KUKA KRL program: MyProgram_067().src

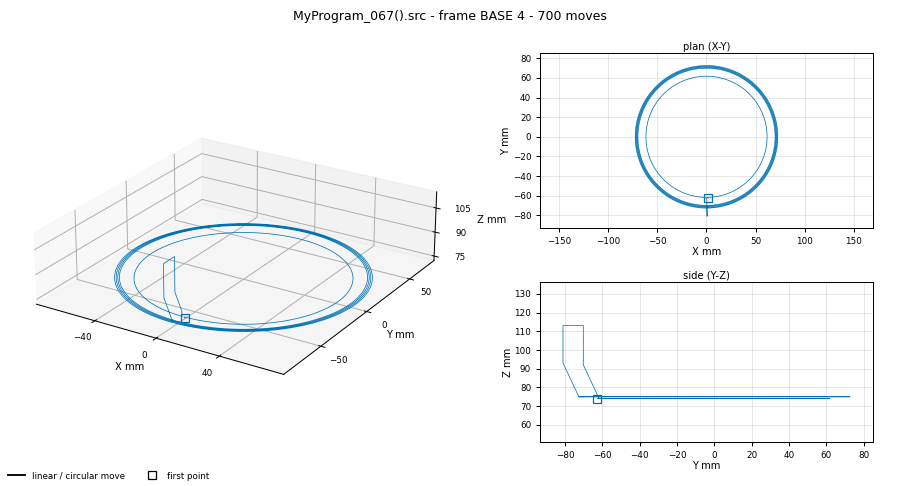
[picture p0: tool path of MyProgram_067().src in frame BASE 4, 700 of 700 moves have a stored position in this frame; points joined in program order, loops and branches not executed]
&ACCESS RVP
&REL 1
&PARAM TEMPLATE = C:\KRC\Roboter\Template\vorgabe
&PARAM EDITMASK = *
DEF MyProgram_067()
; ---- Setting reference (Base) ----
$BASE = BASE_DATA[4]

; --------------------------
; ---- Setting tool (TCP) ----
$TOOL = TOOL_DATA[3]
; --------------------------

$VEL.CP = VEL_APROX_PRINT
Startdeposition()
$VEL.CP = VEL_PRINT
LIN {X 1.6603,Y -62.6279,Z 74,A -94.6717,B 24.8978,C -2.3339,E1 25.0027,E2 178.7795} C_DIS
LIN {X 1.6603,Y -62.6279,Z 74,A -94.6717,B 24.8978,C -2.3339,E1 25.0027,E2 178.7795} C_DIS
Enddeposition()
LIN {X 0.3854,Y -61.7225,Z 74,A -95.5899,B 24.8959,C -2.3553,E1 25.0003,E2 179.6469} C_DIS
Startdeposition()
$VEL.CP = VEL_PRINT
LIN {X 2.2389,Y -61.6864,Z 74,A -92.854,B 24.8939,C -2.3781,E1 25.0081,E2 176.8573} C_DIS
LIN {X 5.2551,Y -61.5029,Z 74,A -90.0412,B 24.8937,C -2.3796,E1 25.0159,E2 174.0424} C_DIS
LIN {X 8.2959,Y -61.1671,Z 74,A -87.2156,B 24.8937,C -2.381,E1 25.0237,E2 171.2156} C_DIS
LIN {X 11.2776,Y -60.6881,Z 74,A -84.42,B 24.8934,C -2.383,E1 25.0314,E2 168.4183} C_DIS
LIN {X 14.2593,Y -60.0576,Z 74,A -81.5934,B 24.8932,C -2.3855,E1 25.0391,E2 165.5894} C_DIS
LIN {X 17.1475,Y -59.2974,Z 74,A -78.8211,B 24.8929,C -2.3885,E1 25.0466,E2 162.8146} C_DIS
LIN {X 20.0481,Y -58.3806,Z 74,A -76.0037,B 24.8927,C -2.3917,E1 25.0541,E2 159.9949} C_DIS
LIN {X 22.9015,Y -57.3215,Z 74,A -73.1974,B 24.8923,C -2.3951,E1 25.0614,E2 157.1866} C_DIS
LIN {X 25.6576,Y -56.1417,Z 74,A -70.4181,B 24.892,C -2.3992,E1 25.0685,E2 154.4046} C_DIS
LIN {X 28.3851,Y -54.8133,Z 74,A -67.6066,B 24.8916,C -2.4037,E1 25.0755,E2 151.5901} C_DIS
LIN {X 31.0814,Y -53.3309,Z 74,A -64.7699,B 24.8912,C -2.4082,E1 25.0824,E2 148.751} C_DIS
LIN {X 33.6554,Y -51.7451,Z 74,A -61.9856,B 24.8907,C -2.413,E1 25.089,E2 145.9645} C_DIS
LIN {X 35.9087,Y -50.2063,Z 74,A -59.347,B 24.89,C -2.4206,E1 25.0951,E2 143.3169} C_DIS
LIN {X 37.9795,Y -48.66,Z 74,A -57.0724,B 24.8899,C -2.4227,E1 25.1001,E2 141.0458} C_DIS
LIN {X 40.2995,Y -46.7566,Z 74,A -54.2947,B 24.8893,C -2.4286,E1 25.106,E2 138.2646} C_DIS
LIN {X 42.5511,Y -44.7173,Z 74,A -51.4857,B 24.8887,C -2.4349,E1 25.1118,E2 135.4522} C_DIS
LIN {X 44.6978,Y -42.5717,Z 74,A -48.6871,B 24.8881,C -2.4413,E1 25.1172,E2 132.6505} C_DIS
LIN {X 46.7261,Y -40.3349,Z 74,A -45.9001,B 24.8875,C -2.448,E1 25.1224,E2 129.8602} C_DIS
LIN {X 48.6424,Y -38.0018,Z 74,A -43.1096,B 24.8869,C -2.455,E1 25.1273,E2 127.0662} C_DIS
LIN {X 50.471,Y -35.5376,Z 74,A -40.2933,B 24.8862,C -2.4619,E1 25.1319,E2 124.2472} C_DIS
LIN {X 52.1299,Y -33.0559,Z 74,A -37.5283,B 24.8855,C -2.4694,E1 25.1361,E2 121.4782} C_DIS
LIN {X 53.7046,Y -30.4313,Z 74,A -34.7004,B 24.8848,C -2.4772,E1 25.1401,E2 118.6466} C_DIS
LIN {X 55.1351,Y -27.7556,Z 74,A -31.916,B 24.8841,C -2.4846,E1 25.1437,E2 115.8594} C_DIS
LIN {X 56.4098,Y -25.0629,Z 74,A -29.1531,B 24.8834,C -2.4927,E1 25.1469,E2 113.0922} C_DIS
LIN {X 57.5735,Y -22.2598,Z 74,A -26.3562,B 24.8826,C -2.5007,E1 25.1498,E2 110.2918} C_DIS
LIN {X 58.5947,Y -19.4131,Z 74,A -23.5811,B 24.8819,C -2.5085,E1 25.1523,E2 107.514} C_DIS
LIN {X 59.4511,Y -16.6049,Z 74,A -20.9319,B 24.8813,C -2.5151,E1 25.1544,E2 104.8645} C_DIS
LIN {X 60.0566,Y -14.2635,Z 74,A -18.6458,B 24.8805,C -2.5231,E1 25.1559,E2 102.5726} C_DIS
LIN {X 60.6831,Y -11.3049,Z 74,A -15.8403,B 24.8797,C -2.5319,E1 25.1574,E2 99.7627} C_DIS
LIN {X 61.1664,Y -8.3014,Z 74,A -13.0483,B 24.8789,C -2.54,E1 25.1586,E2 96.9679} C_DIS
LIN {X 61.4957,Y -5.3376,Z 74,A -10.2981,B 24.8781,C -2.5483,E1 25.1593,E2 94.2143} C_DIS
LIN {X 61.6847,Y -2.2864,Z 74,A -7.4845,B 24.8773,C -2.5567,E1 25.1597,E2 91.3975} C_DIS
LIN {X 61.7226,Y 0.753,Z 74,A -4.6831,B 24.8765,C -2.5652,E1 25.1597,E2 88.5929} C_DIS
LIN {X 61.613,Y 3.7495,Z 74,A -1.9141,B 24.8757,C -2.5736,E1 25.1594,E2 85.8205} C_DIS
LIN {X 61.3515,Y 6.7991,Z 74,A 0.9072,B 24.8748,C -2.582,E1 25.1586,E2 82.9961} C_DIS
LIN {X 60.9452,Y 9.7941,Z 74,A 3.6994,B 24.874,C -2.5903,E1 25.1574,E2 80.2006} C_DIS
LIN {X 60.3961,Y 12.7486,Z 74,A 6.4727,B 24.8732,C -2.5985,E1 25.1559,E2 77.4242} C_DIS
LIN {X 59.69,Y 15.7273,Z 74,A 9.2777,B 24.8725,C -2.6061,E1 25.154,E2 74.6173} C_DIS
LIN {X 58.8596,Y 18.5946,Z 74,A 12.0434,B 24.8717,C -2.6142,E1 25.1518,E2 71.8482} C_DIS
LIN {X 57.8593,Y 21.507,Z 74,A 14.8896,B 24.8709,C -2.6222,E1 25.1491,E2 68.9991} C_DIS
LIN {X 56.7304,Y 24.3291,Z 74,A 17.68,B 24.8702,C -2.6295,E1 25.1461,E2 66.2068} C_DIS
LIN {X 55.4727,Y 27.0745,Z 74,A 20.4596,B 24.8695,C -2.6366,E1 25.1428,E2 63.4253} C_DIS
LIN {X 54.1001,Y 29.7219,Z 74,A 23.2284,B 24.8687,C -2.6441,E1 25.1391,E2 60.6533} C_DIS
LIN {X 52.5629,Y 32.3632,Z 74,A 26.0462,B 24.868,C -2.6511,E1 25.1351,E2 57.8335} C_DIS
LIN {X 50.9005,Y 34.9197,Z 74,A 28.8466,B 24.8674,C -2.6574,E1 25.1307,E2 55.032} C_DIS
LIN {X 49.1544,Y 37.3371,Z 74,A 31.6173,B 24.8667,C -2.6642,E1 25.1261,E2 52.2586} C_DIS
LIN {X 47.2479,Y 39.7224,Z 74,A 34.4307,B 24.8661,C -2.6703,E1 25.1211,E2 49.4438} C_DIS
LIN {X 45.245,Y 41.9895,Z 74,A 37.2149,B 24.8655,C -2.6759,E1 25.1159,E2 46.6586} C_DIS
LIN {X 43.1689,Y 44.1207,Z 74,A 39.9738,B 24.865,C -2.6816,E1 25.1105,E2 43.8978} C_DIS
LIN {X 40.866,Y 46.2623,Z 74,A 42.8566,B 24.8645,C -2.6865,E1 25.1045,E2 41.0151} C_DIS
LIN {X 38.5801,Y 48.1852,Z 74,A 45.6354,B 24.8639,C -2.6918,E1 25.0985,E2 38.2344} C_DIS
LIN {X 36.1981,Y 49.9991,Z 74,A 48.4152,B 24.8634,C -2.6966,E1 25.0923,E2 35.4531} C_DIS
LIN {X 33.6858,Y 51.7251,Z 74,A 51.2263,B 24.863,C -2.7006,E1 25.0857,E2 32.6418} C_DIS
LIN {X 31.0844,Y 53.3292,Z 74,A 54.0465,B 24.8626,C -2.7044,E1 25.079,E2 29.8214} C_DIS
LIN {X 28.4548,Y 54.7773,Z 74,A 56.8332,B 24.8623,C -2.7081,E1 25.0721,E2 27.034} C_DIS
LIN {X 25.7053,Y 56.1203,Z 74,A 59.6662,B 24.862,C -2.7112,E1 25.065,E2 24.2008} C_DIS
LIN {X 22.9276,Y 57.3111,Z 74,A 62.4652,B 24.8617,C -2.714,E1 25.0577,E2 21.4018} C_DIS
LIN {X 20.125,Y 58.3541,Z 74,A 65.2331,B 24.8614,C -2.7162,E1 25.0505,E2 18.6341} C_DIS
LIN {X 17.2286,Y 59.2739,Z 74,A 68.0604,B 24.8612,C -2.7184,E1 25.0429,E2 15.8067} C_DIS
LIN {X 14.2598,Y 60.0575,Z 74,A 70.8892,B 24.8611,C -2.7196,E1 25.0353,E2 12.9792} C_DIS
LIN {X 11.3005,Y 60.684,Z 74,A 73.7045,B 24.861,C -2.721,E1 25.0275,E2 10.1642} C_DIS
LIN {X 8.3143,Y 61.1646,Z 74,A 76.5104,B 24.8609,C -2.7217,E1 25.0198,E2 7.3591} C_DIS
LIN {X 5.3318,Y 61.4963,Z 74,A 79.2951,B 24.8609,C -2.722,E1 25.0121,E2 4.5754} C_DIS
LIN {X 2.2751,Y 61.6852,Z 74,A 82.1298,B 24.8609,C -2.7217,E1 25.0042,E2 1.7423} C_DIS
LIN {X -0.7492,Y 61.7226,Z 74,A 84.9385,B 24.8609,C -2.7212,E1 24.9963,E2 -1.0651} C_DIS
LIN {X -3.7534,Y 61.6128,Z 74,A 87.7403,B 24.861,C -2.7205,E1 24.9885,E2 -3.8658} C_DIS
LIN {X -6.8036,Y 61.3511,Z 74,A 90.5853,B 24.8611,C -2.7191,E1 24.9806,E2 -6.7091} C_DIS
LIN {X -9.7997,Y 60.9443,Z 74,A 93.3961,B 24.8613,C -2.7173,E1 24.9729,E2 -9.5181} C_DIS
LIN {X -12.7347,Y 60.399,Z 74,A 96.1815,B 24.8615,C -2.7154,E1 24.9652,E2 -12.3021} C_DIS
LIN {X -15.7307,Y 59.6891,Z 74,A 99.0339,B 24.8618,C -2.7126,E1 24.9575,E2 -15.1517} C_DIS
LIN {X -18.6193,Y 58.8519,Z 74,A 101.8354,B 24.8621,C -2.7097,E1 24.95,E2 -17.9511} C_DIS
LIN {X -21.5107,Y 57.8579,Z 74,A 104.6799,B 24.8625,C -2.7063,E1 24.9426,E2 -20.7932} C_DIS
LIN {X -24.3152,Y 56.7364,Z 74,A 107.495,B 24.8628,C -2.7026,E1 24.9353,E2 -23.6059} C_DIS
LIN {X -27.0608,Y 55.4793,Z 74,A 110.298,B 24.8633,C -2.6983,E1 24.9282,E2 -26.4059} C_DIS
LIN {X -29.7396,Y 54.0905,Z 74,A 113.118,B 24.8637,C -2.6941,E1 24.9213,E2 -29.2236} C_DIS
LIN {X -32.3962,Y 52.5425,Z 74,A 115.9816,B 24.8642,C -2.6891,E1 24.9144,E2 -32.0842} C_DIS
LIN {X -34.9253,Y 50.8966,Z 74,A 118.787,B 24.8647,C -2.6839,E1 24.9079,E2 -34.8863} C_DIS
LIN {X -37.3715,Y 49.1285,Z 74,A 121.6084,B 24.8653,C -2.6785,E1 24.9016,E2 -37.705} C_DIS
LIN {X -39.7131,Y 47.2556,Z 74,A 124.4197,B 24.8658,C -2.6731,E1 24.8956,E2 -40.514} C_DIS
LIN {X -42.02,Y 45.2168,Z 74,A 127.2728,B 24.8665,C -2.6665,E1 24.8897,E2 -43.3628} C_DIS
LIN {X -44.1641,Y 43.125,Z 74,A 130.0821,B 24.8671,C -2.6605,E1 24.8841,E2 -46.1696} C_DIS
LIN {X -46.2286,Y 40.9042,Z 74,A 132.9067,B 24.8678,C -2.6537,E1 24.8788,E2 -48.9906} C_DIS
LIN {X -48.1786,Y 38.5882,Z 74,A 135.7462,B 24.8684,C -2.6471,E1 24.8738,E2 -51.8273} C_DIS
LIN {X -50.0053,Y 36.1897,Z 74,A 138.5606,B 24.8691,C -2.6399,E1 24.8691,E2 -54.6383} C_DIS
LIN {X -51.7358,Y 33.6696,Z 74,A 141.4276,B 24.8699,C -2.6327,E1 24.8647,E2 -57.5024} C_DIS
LIN {X -53.3279,Y 31.0865,Z 74,A 144.2266,B 24.8707,C -2.6245,E1 24.8607,E2 -60.2961} C_DIS
LIN {X -54.7373,Y 28.5307,Z 74,A 146.9486,B 24.8714,C -2.6169,E1 24.8571,E2 -63.0145} C_DIS
LIN {X -56.0379,Y 25.8822,Z 74,A 149.7819,B 24.872,C -2.6106,E1 24.8537,E2 -65.8481} C_DIS
LIN {X -57.3141,Y 22.9202,Z 74,A 152.7404,B 24.873,C -2.601,E1 24.8505,E2 -68.8} C_DIS
LIN {X -58.3546,Y 20.1234,Z 74,A 155.5303,B 24.8738,C -2.593,E1 24.8479,E2 -71.5865} C_DIS
LIN {X -59.2693,Y 17.2441,Z 74,A 158.3637,B 24.8746,C -2.5849,E1 24.8456,E2 -74.4169} C_DIS
LIN {X -60.0108,Y 14.4512,Z 74,A 161.1191,B 24.8752,C -2.5779,E1 24.8437,E2 -77.1716} C_DIS
LIN {X -60.6856,Y 11.2914,Z 74,A 164.0763,B 24.8762,C -2.5677,E1 24.8421,E2 -80.122} C_DIS
LIN {X -61.1659,Y 8.3053,Z 74,A 166.9043,B 24.877,C -2.5592,E1 24.841,E2 -82.9465} C_DIS
LIN {X -61.4958,Y 5.3368,Z 74,A 169.6974,B 24.8779,C -2.5508,E1 24.8402,E2 -85.7364} C_DIS
LIN {X -61.6838,Y 2.3093,Z 74,A 172.5358,B 24.8787,C -2.5423,E1 24.8398,E2 -88.5716} C_DIS
LIN {X -61.7234,Y -0.6427,Z 74,A 174.9824,B 24.88,C -2.5283,E1 24.8398,E2 -90.9993} C_DIS
LIN {X -61.6544,Y -2.9918,Z 74,A 177.5004,B 24.88,C -2.5276,E1 24.8401,E2 -93.5309} C_DIS
LIN {X -61.4303,Y -6.0469,Z 74,A -179.6505,B 24.8809,C -2.5188,E1 24.8408,E2 -96.376} C_DIS
LIN {X -61.0638,Y -9.0239,Z 74,A -176.8408,B 24.8817,C -2.5106,E1 24.8418,E2 -99.183} C_DIS
LIN {X -60.5483,Y -12.0051,Z 74,A -174.0035,B 24.8824,C -2.5026,E1 24.8433,E2 -102.0179} C_DIS
LIN {X -59.8873,Y -14.9575,Z 74,A -171.1785,B 24.8832,C -2.4944,E1 24.8451,E2 -104.8399} C_DIS
LIN {X -59.0657,Y -17.9298,Z 74,A -168.3034,B 24.884,C -2.4861,E1 24.8473,E2 -107.7118} C_DIS
LIN {X -58.1191,Y -20.7947,Z 74,A -165.4927,B 24.8847,C -2.4781,E1 24.8499,E2 -110.5194} C_DIS
LIN {X -57.0415,Y -23.59,Z 74,A -162.6844,B 24.8854,C -2.4707,E1 24.8528,E2 -113.3257} C_DIS
LIN {X -55.8177,Y -26.3552,Z 74,A -159.8503,B 24.8861,C -2.4634,E1 24.8561,E2 -116.1578} C_DIS
LIN {X -54.4463,Y -29.0833,Z 74,A -157.0013,B 24.8868,C -2.456,E1 24.8597,E2 -119.0044} C_DIS
LIN {X -52.9641,Y -31.702,Z 74,A -154.1929,B 24.8874,C -2.449,E1 24.8637,E2 -121.8106} C_DIS
LIN {X -51.3391,Y -34.2714,Z 74,A -151.3597,B 24.8881,C -2.4421,E1 24.868,E2 -124.6415} C_DIS
LIN {X -49.6548,Y -36.6683,Z 74,A -148.7218,B 24.8888,C -2.4339,E1 24.8723,E2 -127.2727} C_DIS
LIN {X -47.9584,Y -38.8599,Z 74,A -146.0482,B 24.8892,C -2.4299,E1 24.8769,E2 -129.9492} C_DIS
LIN {X -45.9944,Y -41.1657,Z 74,A -143.4282,B 24.8901,C -2.4198,E1 24.8817,E2 -132.5572} C_DIS
LIN {X -44.1975,Y -43.0907,Z 74,A -140.7574,B 24.8901,C -2.419,E1 24.8869,E2 -135.2376} C_DIS
LIN {X -42.0309,Y -45.2066,Z 74,A -137.9338,B 24.8907,C -2.4136,E1 24.8926,E2 -138.06} C_DIS
LIN {X -39.7422,Y -47.2314,Z 74,A -135.0869,B 24.8911,C -2.4084,E1 24.8986,E2 -140.9056} C_DIS
LIN {X -37.3852,Y -49.118,Z 74,A -132.2786,B 24.8916,C -2.4036,E1 24.9048,E2 -143.7127} C_DIS
LIN {X -34.9404,Y -50.8862,Z 74,A -129.4612,B 24.892,C -2.3994,E1 24.9112,E2 -146.5297} C_DIS
LIN {X -32.3849,Y -52.5496,Z 74,A -126.6115,B 24.8923,C -2.3955,E1 24.9179,E2 -149.3793} C_DIS
LIN {X -29.7939,Y -54.0606,Z 74,A -123.8249,B 24.8927,C -2.3918,E1 24.9247,E2 -152.1652} C_DIS
LIN {X -27.1134,Y -55.4534,Z 74,A -121.0032,B 24.8929,C -2.3887,E1 24.9317,E2 -154.9871} C_DIS
LIN {X -24.3297,Y -56.7301,Z 74,A -118.1616,B 24.8932,C -2.3856,E1 24.939,E2 -157.8282} C_DIS
LIN {X -21.5259,Y -57.8521,Z 74,A -115.3559,B 24.8934,C -2.3831,E1 24.9463,E2 -160.6338} C_DIS
LIN {X -18.6841,Y -58.8313,Z 74,A -112.5554,B 24.8936,C -2.3811,E1 24.9537,E2 -163.4348} C_DIS
LIN {X -15.7315,Y -59.6889,Z 74,A -109.7003,B 24.8938,C -2.3794,E1 24.9614,E2 -166.2902} C_DIS
LIN {X -12.8257,Y -60.3798,Z 74,A -106.9156,B 24.8938,C -2.3783,E1 24.969,E2 -169.076} C_DIS
LIN {X -9.8156,Y -60.9417,Z 74,A -104.0755,B 24.8939,C -2.3774,E1 24.9768,E2 -171.9166} C_DIS
LIN {X -6.804,Y -61.3511,Z 74,A -101.2661,B 24.894,C -2.3767,E1 24.9846,E2 -174.7263} C_DIS
LIN {X -3.8288,Y -61.6081,Z 74,A -98.4765,B 24.894,C -2.3771,E1 24.9924,E2 -177.518} C_DIS
LIN {X -0.7696,Y -61.7223,Z 74,A -95.6423,B 24.894,C -2.3773,E1 25.0003,E2 -180.3531} C_DIS
LIN {X -0.7696,Y -61.7223,Z 74,A -95.6423,B 24.894,C -2.3773,E1 25.0003,E2 -180.3531} C_DIS
Enddeposition()
LIN {X 0.385,Y -63.8356,Z 78.5315,A -95.5798,B 24.8963,C -2.351,E1 25.0003,E2 -180.3531} C_DIS
LIN {X 0.384,Y -70.1749,Z 92.1262,A -95.5544,B 24.8972,C -2.3403,E1 25.0003,E2 -180.3531} C_DIS
LIN {X 0.384,Y -70.1749,Z 113.1262,A -95.9113,B 24.8836,C -2.4906,E1 25.0003,E2 -180.3531} C_DIS
LIN {X 0.598,Y -81.0561,Z 113.1262,A -94.7572,B 24.8982,C -2.3288,E1 25.0024,E2 -181.1228} C_DIS
LIN {X 0.598,Y -81.0561,Z 93.1262,A -94.4172,B 24.9104,C -2.1856,E1 25.0024,E2 -181.1228} C_DIS
LIN {X 0.5139,Y -74.7174,Z 79.5315,A -94.4404,B 24.9096,C -2.1954,E1 25.0024,E2 -181.1228} C_DIS
LIN {X 0.4859,Y -72.6045,Z 75,A -94.4497,B 24.9093,C -2.1993,E1 25.0024,E2 -181.1228} C_DIS
Startdeposition()
$VEL.CP = VEL_PRINT
LIN {X -2.6725,Y -72.56,Z 75,A -97.8407,B 24.9112,C -2.1754,E1 24.9928,E2 -177.6748} C_DIS
LIN {X -5.5896,Y -72.3926,Z 75,A -100.1329,B 24.9112,C -2.1757,E1 24.9864,E2 -175.3826} C_DIS
LIN {X -8.6409,Y -72.0921,Z 75,A -102.5384,B 24.9112,C -2.1764,E1 24.9797,E2 -172.9772} C_DIS
LIN {X -11.5346,Y -71.6872,Z 75,A -104.9376,B 24.9113,C -2.1745,E1 24.9731,E2 -170.5715} C_DIS
LIN {X -14.1654,Y -71.214,Z 75,A -107.0488,B 24.9113,C -2.1753,E1 24.9673,E2 -168.4598} C_DIS
LIN {X -16.7769,Y -70.6444,Z 75,A -109.1605,B 24.9112,C -2.1762,E1 24.9616,E2 -166.3476} C_DIS
LIN {X -19.3658,Y -69.979,Z 75,A -111.2729,B 24.9111,C -2.1774,E1 24.9559,E2 -164.2349} C_DIS
LIN {X -21.9284,Y -69.2188,Z 75,A -113.3855,B 24.911,C -2.1788,E1 24.9502,E2 -162.122} C_DIS
LIN {X -24.4613,Y -68.3648,Z 75,A -115.4988,B 24.9108,C -2.1805,E1 24.9447,E2 -160.0085} C_DIS
LIN {X -26.961,Y -67.4181,Z 75,A -117.6126,B 24.9107,C -2.1824,E1 24.9392,E2 -157.8946} C_DIS
LIN {X -29.4242,Y -66.38,Z 75,A -119.5937,B 24.9102,C -2.1877,E1 24.9341,E2 -155.9216} C_DIS
LIN {X -31.8476,Y -65.252,Z 75,A -121.8419,B 24.9103,C -2.1868,E1 24.9284,E2 -153.6654} C_DIS
LIN {X -34.4465,Y -63.9169,Z 75,A -124.0765,B 24.9099,C -2.1915,E1 24.9229,E2 -151.4358} C_DIS
LIN {X -37.1143,Y -62.4056,Z 75,A -126.3435,B 24.9093,C -2.1985,E1 24.9175,E2 -149.1788} C_DIS
LIN {X -39.0552,Y -61.2097,Z 75,A -128.3088,B 24.9094,C -2.1972,E1 24.9128,E2 -147.2042} C_DIS
LIN {X -41.2817,Y -59.7307,Z 75,A -130.4258,B 24.9092,C -2.2004,E1 24.9079,E2 -145.0877} C_DIS
LIN {X -43.4522,Y -58.1708,Z 75,A -132.5433,B 24.9089,C -2.2038,E1 24.9031,E2 -142.9708} C_DIS
LIN {X -45.8694,Y -56.2844,Z 75,A -134.8122,B 24.9082,C -2.2117,E1 24.8982,E2 -140.7123} C_DIS
LIN {X -47.91,Y -54.5579,Z 75,A -136.9308,B 24.9079,C -2.2155,E1 24.8937,E2 -138.5945} C_DIS
LIN {X -49.8857,Y -52.7575,Z 75,A -139.0494,B 24.9076,C -2.2194,E1 24.8893,E2 -136.4767} C_DIS
LIN {X -51.7937,Y -50.8856,Z 75,A -141.1686,B 24.9073,C -2.2236,E1 24.8852,E2 -134.3584} C_DIS
LIN {X -53.6316,Y -48.9447,Z 75,A -143.4337,B 24.9072,C -2.2245,E1 24.8808,E2 -132.0856} C_DIS
LIN {X -55.5582,Y -46.7481,Z 75,A -145.818,B 24.9069,C -2.2279,E1 24.8765,E2 -129.6985} C_DIS
LIN {X -57.3931,Y -44.4743,Z 75,A -148.0842,B 24.9064,C -2.2342,E1 24.8726,E2 -127.4368} C_DIS
LIN {X -59.2196,Y -42.0116,Z 75,A -150.5022,B 24.9059,C -2.2401,E1 24.8686,E2 -125.0212} C_DIS
LIN {X -60.8628,Y -39.5956,Z 75,A -152.9141,B 24.9056,C -2.2435,E1 24.8649,E2 -122.6053} C_DIS
LIN {X -62.4056,Y -37.1143,Z 75,A -155.1552,B 24.9049,C -2.251,E1 24.8616,E2 -120.3705} C_DIS
LIN {X -63.9169,Y -34.4465,Z 75,A -157.5744,B 24.9044,C -2.2574,E1 24.8583,E2 -117.954} C_DIS
LIN {X -65.252,Y -31.8476,Z 75,A -159.9875,B 24.9041,C -2.2613,E1 24.8553,E2 -115.5371} C_DIS
LIN {X -66.38,Y -29.4242,Z 75,A -161.9261,B 24.9032,C -2.271,E1 24.8531,E2 -113.6111} C_DIS
LIN {X -67.4181,Y -26.961,Z 75,A -164.2138,B 24.9031,C -2.273,E1 24.8507,E2 -111.3155} C_DIS
LIN {X -68.4472,Y -24.2265,Z 75,A -166.4758,B 24.9024,C -2.2807,E1 24.8485,E2 -109.059} C_DIS
LIN {X -69.409,Y -21.3151,Z 75,A -168.7509,B 24.9015,C -2.2911,E1 24.8466,E2 -106.7957} C_DIS
LIN {X -70.1465,Y -18.7459,Z 75,A -171.0203,B 24.9013,C -2.2938,E1 24.8449,E2 -104.5197} C_DIS
LIN {X -70.8449,Y -15.9088,Z 75,A -173.435,B 24.9009,C -2.2984,E1 24.8433,E2 -102.1017} C_DIS
LIN {X -71.4266,Y -13.0454,Z 75,A -175.6787,B 24.9002,C -2.3069,E1 24.8421,E2 -99.8649} C_DIS
LIN {X -71.9136,Y -10.0182,Z 75,A -178.1001,B 24.8995,C -2.3143,E1 24.8411,E2 -97.447} C_DIS
LIN {X -72.2596,Y -7.1169,Z 75,A 179.4846,B 24.8991,C -2.3191,E1 24.8404,E2 -95.0286} C_DIS
LIN {X -72.4726,Y -4.4524,Z 75,A 177.4944,B 24.8983,C -2.3283,E1 24.84,E2 -93.0486} C_DIS
LIN {X -72.5873,Y -1.7819,Z 75,A 175.2122,B 24.898,C -2.3312,E1 24.8398,E2 -90.7594} C_DIS
LIN {X -72.5873,Y 1.7819,Z 75,A 172.4034,B 24.8972,C -2.3402,E1 24.8398,E2 -87.9551} C_DIS
LIN {X -72.4726,Y 4.4524,Z 75,A 170.4127,B 24.8964,C -2.3495,E1 24.8402,E2 -85.9747} C_DIS
LIN {X -72.2596,Y 7.1169,Z 75,A 168.1543,B 24.8961,C -2.3529,E1 24.8407,E2 -83.7109} C_DIS
LIN {X -71.9136,Y 10.0182,Z 75,A 165.9103,B 24.8954,C -2.3616,E1 24.8415,E2 -81.4742} C_DIS
LIN {X -71.4266,Y 13.0454,Z 75,A 163.6341,B 24.8944,C -2.3724,E1 24.8426,E2 -79.2103} C_DIS
LIN {X -70.898,Y 15.6656,Z 75,A 161.5098,B 24.8938,C -2.3787,E1 24.8438,E2 -77.0886} C_DIS
LIN {X -70.3937,Y 17.7964,Z 75,A 159.5628,B 24.8938,C -2.3792,E1 24.8451,E2 -75.1315} C_DIS
LIN {X -69.5535,Y 20.8387,Z 75,A 157.2614,B 24.8927,C -2.3911,E1 24.8469,E2 -72.8452} C_DIS
LIN {X -68.83,Y 23.1158,Z 75,A 155.2541,B 24.8924,C -2.3942,E1 24.8486,E2 -70.8338} C_DIS
LIN {X -67.832,Y 25.8989,Z 75,A 152.8679,B 24.8919,C -2.4002,E1 24.8509,E2 -68.4482} C_DIS
LIN {X -66.7361,Y 28.6074,Z 75,A 150.4533,B 24.8915,C -2.4046,E1 24.8535,E2 -66.031} C_DIS
LIN {X -65.5301,Y 31.2688,Z 75,A 148.2102,B 24.8907,C -2.4129,E1 24.8561,E2 -63.7953} C_DIS
LIN {X -64.1516,Y 34.0075,Z 75,A 145.9355,B 24.8898,C -2.4231,E1 24.859,E2 -61.5329} C_DIS
LIN {X -62.8564,Y 36.3457,Z 75,A 143.8125,B 24.8893,C -2.4289,E1 24.8619,E2 -59.4125} C_DIS
LIN {X -61.476,Y 38.6347,Z 75,A 141.7013,B 24.8887,C -2.4347,E1 24.865,E2 -57.3044} C_DIS
LIN {X -60.2328,Y 40.5456,Z 75,A 139.7188,B 24.8887,C -2.4356,E1 24.8681,E2 -55.314} C_DIS
LIN {X -58.4673,Y 43.0524,Z 75,A 137.4451,B 24.8878,C -2.4454,E1 24.8717,E2 -53.0527} C_DIS
LIN {X -56.843,Y 45.1753,Z 75,A 135.3232,B 24.8873,C -2.4506,E1 24.8754,E2 -50.9332} C_DIS
LIN {X -55.3968,Y 46.9375,Z 75,A 133.3533,B 24.8873,C -2.4513,E1 24.8789,E2 -48.9559} C_DIS
LIN {X -53.3657,Y 49.2345,Z 75,A 131.0807,B 24.8864,C -2.4607,E1 24.8831,E2 -46.6956} C_DIS
LIN {X -51.5174,Y 51.1654,Z 75,A 128.8185,B 24.8862,C -2.4623,E1 24.8875,E2 -44.4274} C_DIS
LIN {X -49.4179,Y 53.1974,Z 75,A 126.537,B 24.8857,C -2.4682,E1 24.8921,E2 -42.1506} C_DIS
LIN {X -47.4264,Y 54.9803,Z 75,A 124.331,B 24.8854,C -2.4707,E1 24.8968,E2 -39.9418} C_DIS
LIN {X -45.3705,Y 56.6887,Z 75,A 122.2974,B 24.8848,C -2.477,E1 24.9012,E2 -37.9155} C_DIS
LIN {X -43.2532,Y 58.3203,Z 75,A 120.0445,B 24.8848,C -2.478,E1 24.9062,E2 -35.657} C_DIS
LIN {X -41.0773,Y 59.8728,Z 75,A 117.9258,B 24.8844,C -2.4819,E1 24.911,E2 -33.5405} C_DIS
LIN {X -38.8457,Y 61.3441,Z 75,A 115.8074,B 24.884,C -2.4857,E1 24.916,E2 -31.4242} C_DIS
LIN {X -36.5615,Y 62.7324,Z 75,A 113.6896,B 24.8837,C -2.4893,E1 24.9211,E2 -29.3085} C_DIS
LIN {X -34.0075,Y 64.1516,Z 75,A 111.453,B 24.8832,C -2.4948,E1 24.9266,E2 -27.0787} C_DIS
LIN {X -31.2688,Y 65.5301,Z 75,A 109.1851,B 24.8825,C -2.5022,E1 24.9322,E2 -24.8225} C_DIS
LIN {X -28.8356,Y 66.6367,Z 75,A 107.0687,B 24.8822,C -2.5051,E1 24.9376,E2 -22.7079} C_DIS
LIN {X -26.3633,Y 67.6528,Z 75,A 104.9559,B 24.8819,C -2.5079,E1 24.9431,E2 -20.5971} C_DIS
LIN {X -24.2265,Y 68.4472,Z 75,A 102.9886,B 24.8821,C -2.5061,E1 24.9483,E2 -18.6217} C_DIS
LIN {X -21.3151,Y 69.409,Z 75,A 100.7228,B 24.8815,C -2.5126,E1 24.9543,E2 -16.3672} C_DIS
LIN {X -18.7459,Y 70.1465,Z 75,A 98.6085,B 24.8813,C -2.5147,E1 24.9599,E2 -14.2545} C_DIS
LIN {X -16.1513,Y 70.7889,Z 75,A 96.4947,B 24.8811,C -2.5165,E1 24.9657,E2 -12.1423} C_DIS
LIN {X -13.921,Y 71.2611,Z 75,A 94.5323,B 24.8814,C -2.514,E1 24.9711,E2 -10.1716} C_DIS
LIN {X -10.8999,Y 71.7853,Z 75,A 92.1237,B 24.8812,C -2.516,E1 24.9777,E2 -7.7654} C_DIS
LIN {X -8.0031,Y 72.1668,Z 75,A 89.8553,B 24.881,C -2.5182,E1 24.984,E2 -5.5008} C_DIS
LIN {X -5.3415,Y 72.4125,Z 75,A 87.611,B 24.8812,C -2.5158,E1 24.9902,E2 -3.2498} C_DIS
LIN {X -2.7078,Y 72.5585,Z 75,A 85.5444,B 24.8811,C -2.5169,E1 24.996,E2 -1.1853} C_DIS
LIN {X 0.2489,Y 72.6077,Z 75,A 83.2706,B 24.8809,C -2.5189,E1 25.0023,E2 1.0838} C_DIS
LIN {X 3.3141,Y 72.5324,Z 75,A 81.01,B 24.8805,C -2.5232,E1 25.0086,E2 3.3337} C_DIS
LIN {X 5.5896,Y 72.3926,Z 75,A 79.0516,B 24.8809,C -2.5191,E1 25.0141,E2 5.301} C_DIS
LIN {X 8.5677,Y 72.1007,Z 75,A 76.6842,B 24.8809,C -2.5186,E1 25.0207,E2 7.6679} C_DIS
LIN {X 11.5346,Y 71.6872,Z 75,A 74.2509,B 24.8812,C -2.5161,E1 25.0274,E2 10.1048} C_DIS
LIN {X 14.1654,Y 71.214,Z 75,A 72.1434,B 24.8812,C -2.5153,E1 25.0332,E2 12.2118} C_DIS
LIN {X 16.7769,Y 70.6444,Z 75,A 70.0365,B 24.8813,C -2.5143,E1 25.0389,E2 14.3183} C_DIS
LIN {X 19.3658,Y 69.979,Z 75,A 67.93,B 24.8815,C -2.513,E1 25.0446,E2 16.4244} C_DIS
LIN {X 21.9284,Y 69.2188,Z 75,A 65.9569,B 24.8813,C -2.515,E1 25.0498,E2 18.3893} C_DIS
LIN {X 24.4613,Y 68.3648,Z 75,A 63.7189,B 24.8818,C -2.5098,E1 25.0557,E2 20.6351} C_DIS
LIN {X 26.961,Y 67.4181,Z 75,A 61.6411,B 24.8818,C -2.5086,E1 25.0611,E2 22.7112} C_DIS
LIN {X 29.4242,Y 66.38,Z 75,A 59.5099,B 24.8821,C -2.5057,E1 25.0666,E2 24.8441} C_DIS
LIN {X 32.1584,Y 65.098,Z 75,A 57.2569,B 24.8821,C -2.5064,E1 25.0723,E2 27.0897} C_DIS
LIN {X 34.7922,Y 63.7294,Z 75,A 54.89,B 24.8824,C -2.5026,E1 25.0781,E2 29.4588} C_DIS
LIN {X 37.3286,Y 62.279,Z 75,A 52.4994,B 24.883,C -2.497,E1 25.0839,E2 31.8553} C_DIS
LIN {X 39.5956,Y 60.8628,Z 75,A 50.3972,B 24.8833,C -2.494,E1 25.0888,E2 33.9579} C_DIS
LIN {X 42.0116,Y 59.2196,Z 75,A 48.1772,B 24.8833,C -2.4925,E1 25.0939,E2 36.1738} C_DIS
LIN {X 44.4743,Y 57.3931,Z 75,A 45.7819,B 24.8837,C -2.4889,E1 25.0992,E2 38.5689} C_DIS
LIN {X 46.7481,Y 55.5582,Z 75,A 43.3936,B 24.8843,C -2.4823,E1 25.1044,E2 40.9637} C_DIS
LIN {X 48.7614,Y 53.7999,Z 75,A 41.2933,B 24.8847,C -2.4785,E1 25.1088,E2 43.0647} C_DIS
LIN {X 50.8287,Y 51.85,Z 75,A 39.0981,B 24.885,C -2.4752,E1 25.1132,E2 45.2587} C_DIS
LIN {X 52.7575,Y 49.8857,Z 75,A 36.9761,B 24.8853,C -2.4719,E1 25.1173,E2 47.3792} C_DIS
LIN {X 54.8166,Y 47.6138,Z 75,A 34.7274,B 24.8853,C -2.4712,E1 25.1215,E2 49.6195} C_DIS
LIN {X 56.532,Y 45.5639,Z 75,A 32.629,B 24.8858,C -2.4666,E1 25.1252,E2 51.719} C_DIS
LIN {X 57.9346,Y 43.7667,Z 75,A 30.6806,B 24.8866,C -2.4582,E1 25.1285,E2 53.6782} C_DIS
LIN {X 59.7307,Y 41.2817,Z 75,A 28.4331,B 24.8866,C -2.457,E1 25.1321,E2 55.9175} C_DIS
LIN {X 61.2097,Y 39.0552,Z 75,A 26.3357,B 24.8872,C -2.452,E1 25.1354,E2 58.0163} C_DIS
LIN {X 62.6057,Y 36.7758,Z 75,A 24.2385,B 24.8876,C -2.4468,E1 25.1384,E2 60.115} C_DIS
LIN {X 63.9169,Y 34.4465,Z 75,A 21.998,B 24.8885,C -2.4375,E1 25.1414,E2 62.3659} C_DIS
LIN {X 65.252,Y 31.8476,Z 75,A 19.6143,B 24.8893,C -2.4289,E1 25.1444,E2 64.7571} C_DIS
LIN {X 66.38,Y 29.4242,Z 75,A 17.6502,B 24.8894,C -2.4271,E1 25.1467,E2 66.7148} C_DIS
LIN {X 67.4181,Y 26.961,Z 75,A 15.4222,B 24.8903,C -2.4177,E1 25.149,E2 68.9527} C_DIS
LIN {X 68.4472,Y 24.2265,Z 75,A 13.2126,B 24.8907,C -2.4137,E1 25.1512,E2 71.1594} C_DIS
LIN {X 69.409,Y 21.3151,Z 75,A 10.9632,B 24.8909,C -2.4114,E1 25.1531,E2 73.4015} C_DIS
LIN {X 70.1221,Y 18.8361,Z 75,A 8.7699,B 24.8918,C -2.4008,E1 25.1547,E2 75.6073} C_DIS
LIN {X 70.8449,Y 15.9088,Z 75,A 6.3421,B 24.8926,C -2.3922,E1 25.1563,E2 78.0414} C_DIS
LIN {X 71.4266,Y 13.0454,Z 75,A 4.1291,B 24.893,C -2.3878,E1 25.1575,E2 80.252} C_DIS
LIN {X 71.8986,Y 10.1243,Z 75,A 1.793,B 24.8937,C -2.3805,E1 25.1584,E2 82.5915} C_DIS
LIN {X 72.2596,Y 7.1169,Z 75,A -0.6405,B 24.8944,C -2.3717,E1 25.1592,E2 85.0312} C_DIS
LIN {X 72.4726,Y 4.4524,Z 75,A -2.6029,B 24.8947,C -2.3693,E1 25.1596,E2 86.9877} C_DIS
LIN {X 72.5873,Y 1.7819,Z 75,A -4.8272,B 24.8956,C -2.3593,E1 25.1598,E2 89.2224} C_DIS
LIN {X 72.5919,Y -1.5331,Z 75,A -7.0063,B 24.8952,C -2.3636,E1 25.1598,E2 91.3783} C_DIS
LIN {X 72.5217,Y -3.5628,Z 75,A -9.0187,B 24.8967,C -2.3467,E1 25.1595,E2 93.4187} C_DIS
LIN {X 72.3186,Y -6.4775,Z 75,A -11.2309,B 24.8971,C -2.3421,E1 25.159,E2 95.6287} C_DIS
LIN {X 71.9806,Y -9.525,Z 75,A -13.6187,B 24.8977,C -2.3353,E1 25.1582,E2 98.0185} C_DIS
LIN {X 71.5402,Y -12.4134,Z 75,A -16.0001,B 24.8985,C -2.3258,E1 25.1571,E2 100.4083} C_DIS
LIN {X 70.9884,Y -15.251,Z 75,A -18.2037,B 24.8989,C -2.3208,E1 25.1559,E2 102.6108} C_DIS
LIN {X 70.2733,Y -18.2645,Z 75,A -20.4571,B 24.8991,C -2.3187,E1 25.1544,E2 104.8562} C_DIS
LIN {X 69.5535,Y -20.8387,Z 75,A -22.5518,B 24.8997,C -2.3125,E1 25.1528,E2 106.9535} C_DIS
LIN {X 68.7393,Y -23.3847,Z 75,A -24.6468,B 24.9002,C -2.3064,E1 25.151,E2 109.051} C_DIS
LIN {X 67.832,Y -25.8989,Z 75,A -26.7417,B 24.9007,C -2.3004,E1 25.1489,E2 111.1485} C_DIS
LIN {X 66.8328,Y -28.3781,Z 75,A -28.8369,B 24.9012,C -2.2944,E1 25.1467,E2 113.2462} C_DIS
LIN {X 65.9089,Y -30.4623,Z 75,A -30.7826,B 24.9021,C -2.2849,E1 25.1445,E2 115.204} C_DIS
LIN {X 64.5641,Y -33.2177,Z 75,A -33.1717,B 24.9026,C -2.2786,E1 25.1415,E2 117.5951} C_DIS
LIN {X 63.1763,Y -35.7889,Z 75,A -35.5545,B 24.9034,C -2.2697,E1 25.1382,E2 119.9865} C_DIS
LIN {X 61.8162,Y -38.09,Z 75,A -37.5185,B 24.9035,C -2.2679,E1 25.1354,E2 121.9447} C_DIS
LIN {X 60.3723,Y -40.3395,Z 75,A -39.6148,B 24.904,C -2.2624,E1 25.1322,E2 124.0436} C_DIS
LIN {X 58.8466,Y -42.5343,Z 75,A -41.7112,B 24.9044,C -2.257,E1 25.1288,E2 126.1425} C_DIS
LIN {X 57.2412,Y -44.6715,Z 75,A -43.9405,B 24.9052,C -2.248,E1 25.125,E2 128.3824} C_DIS
LIN {X 55.5582,Y -46.7481,Z 75,A -46.0376,B 24.9056,C -2.2429,E1 25.1213,E2 130.482} C_DIS
LIN {X 53.7999,Y -48.7614,Z 75,A -48.1351,B 24.906,C -2.2379,E1 25.1174,E2 132.5819} C_DIS
LIN {X 51.9686,Y -50.7085,Z 75,A -50.2058,B 24.9064,C -2.2338,E1 25.1134,E2 134.6534} C_DIS
LIN {X 50.067,Y -52.587,Z 75,A -52.3313,B 24.9068,C -2.2284,E1 25.1091,E2 136.7829} C_DIS
LIN {X 47.91,Y -54.5579,Z 75,A -54.5482,B 24.9071,C -2.2256,E1 25.1045,E2 138.9974} C_DIS
LIN {X 45.4981,Y -56.5853,Z 75,A -56.9878,B 24.9074,C -2.2215,E1 25.0992,E2 141.4376} C_DIS
LIN {X 43.2532,Y -58.3203,Z 75,A -59.3282,B 24.9081,C -2.2139,E1 25.094,E2 143.7874} C_DIS
LIN {X 40.8712,Y -60.0123,Z 75,A -61.5465,B 24.9082,C -2.2118,E1 25.0889,E2 146.0031} C_DIS
LIN {X 38.3011,Y -61.6844,Z 75,A -63.7971,B 24.9082,C -2.2118,E1 25.0836,E2 148.2463} C_DIS
LIN {X 36.1505,Y -62.9686,Z 75,A -65.8241,B 24.9086,C -2.2069,E1 25.0787,E2 150.2789} C_DIS
LIN {X 34.0075,Y -64.1516,Z 75,A -67.849,B 24.9091,C -2.201,E1 25.0738,E2 152.3118} C_DIS
LIN {X 31.2827,Y -65.5234,Z 75,A -70.0935,B 24.9091,C -2.2016,E1 25.0681,E2 154.5489} C_DIS
LIN {X 28.8356,Y -66.6367,Z 75,A -72.2035,B 24.9093,C -2.1987,E1 25.0628,E2 156.6605} C_DIS
LIN {X 26.3633,Y -67.6529,Z 75,A -74.3059,B 24.9095,C -2.1959,E1 25.0573,E2 158.7648} C_DIS
LIN {X 24.2265,Y -68.4472,Z 75,A -76.259,B 24.9101,C -2.1894,E1 25.0522,E2 160.7293} C_DIS
LIN {X 21.3151,Y -69.409,Z 75,A -78.5132,B 24.91,C -2.191,E1 25.0462,E2 162.9755} C_DIS
LIN {X 18.7459,Y -70.1465,Z 75,A -80.7618,B 24.9105,C -2.185,E1 25.0401,E2 165.2347} C_DIS
LIN {X 15.9088,Y -70.8449,Z 75,A -83.1476,B 24.9108,C -2.1806,E1 25.0336,E2 167.6274} C_DIS
LIN {X 13.0454,Y -71.4266,Z 75,A -85.3792,B 24.9108,C -2.1807,E1 25.0275,E2 169.8562} C_DIS
LIN {X 10.0182,Y -71.9136,Z 75,A -87.78,B 24.9108,C -2.1795,E1 25.0209,E2 172.2575} C_DIS
LIN {X 7.1169,Y -72.2596,Z 75,A -90.1752,B 24.9112,C -2.1758,E1 25.0142,E2 174.6599} C_DIS
LIN {X 4.4524,Y -72.4726,Z 75,A -92.1495,B 24.911,C -2.1784,E1 25.0087,E2 176.6272} C_DIS
LIN {X 1.7819,Y -72.5873,Z 75,A -94.3902,B 24.9113,C -2.1743,E1 25.0024,E2 178.8771} C_DIS
LIN {X 1.7819,Y -72.5873,Z 75,A -94.3902,B 24.9113,C -2.1743,E1 25.0024,E2 178.8771} C_DIS
Enddeposition()
LIN {X 0.4761,Y -71.7039,Z 75,A -94.6132,B 24.9083,C -2.2107,E1 25.0021,E2 179.0138} C_DIS
Startdeposition()
$VEL.CP = VEL_PRINT
LIN {X 3.0911,Y -71.6418,Z 75,A -92.1776,B 24.9075,C -2.2203,E1 25.0089,E2 176.5557} C_DIS
LIN {X 6.19,Y -71.4419,Z 75,A -89.6697,B 24.9074,C -2.2222,E1 25.0159,E2 174.0447} C_DIS
LIN {X 9.4285,Y -71.0862,Z 75,A -87.0576,B 24.9072,C -2.224,E1 25.0232,E2 171.4303} C_DIS
LIN {X 12.5111,Y -70.6088,Z 75,A -84.5359,B 24.907,C -2.2267,E1 25.0301,E2 168.9048} C_DIS
LIN {X 15.7853,Y -69.9504,Z 75,A -81.9657,B 24.907,C -2.2264,E1 25.0371,E2 166.3386} C_DIS
LIN {X 17.8363,Y -69.4547,Z 75,A -80.2161,B 24.9067,C -2.2298,E1 25.0419,E2 164.5835} C_DIS
LIN {X 20.9995,Y -68.5651,Z 75,A -77.1541,B 24.9055,C -2.2446,E1 25.0501,E2 161.4919} C_DIS
LIN {X 25.166,Y -67.1478,Z 75,A -74.1453,B 24.9063,C -2.2353,E1 25.058,E2 158.5113} C_DIS
LIN {X 28.269,Y -65.9025,Z 75,A -71.4501,B 24.9059,C -2.2397,E1 25.0649,E2 155.8118} C_DIS
LIN {X 31.7177,Y -64.3126,Z 75,A -68.4955,B 24.9057,C -2.2423,E1 25.0724,E2 152.8588} C_DIS
LIN {X 34.5476,Y -62.8389,Z 75,A -65.8568,B 24.9051,C -2.2491,E1 25.0789,E2 150.2116} C_DIS
LIN {X 37.1045,Y -61.3627,Z 75,A -63.6241,B 24.9051,C -2.2498,E1 25.0843,E2 147.9838} C_DIS
LIN {X 39.8697,Y -59.6043,Z 75,A -60.8762,B 24.9043,C -2.2585,E1 25.0907,E2 145.2245} C_DIS
LIN {X 42.7046,Y -57.6065,Z 75,A -58.2413,B 24.9042,C -2.2603,E1 25.0967,E2 142.5945} C_DIS
LIN {X 44.6014,Y -56.1502,Z 75,A -56.3052,B 24.9037,C -2.2651,E1 25.1009,E2 140.6542} C_DIS
LIN {X 46.7728,Y -54.3556,Z 75,A -54.0231,B 24.9032,C -2.271,E1 25.1058,E2 138.3671} C_DIS
LIN {X 49.0765,Y -52.2839,Z 75,A -51.597,B 24.9029,C -2.2754,E1 25.1108,E2 135.9405} C_DIS
LIN {X 51.2433,Y -50.1629,Z 75,A -49.1218,B 24.9022,C -2.2827,E1 25.1157,E2 133.4585} C_DIS
LIN {X 53.2897,Y -47.9827,Z 75,A -46.8331,B 24.902,C -2.2858,E1 25.12,E2 131.1725} C_DIS
LIN {X 55.4453,Y -45.4762,Z 75,A -44.1098,B 24.9012,C -2.2949,E1 25.1249,E2 128.4402} C_DIS
LIN {X 57.1838,Y -43.2686,Z 75,A -41.9145,B 24.9008,C -2.2994,E1 25.1287,E2 126.2445} C_DIS
LIN {X 59.0271,Y -40.718,Z 75,A -39.4512,B 24.9003,C -2.3048,E1 25.1326,E2 123.7805} C_DIS
LIN {X 60.6496,Y -38.26,Z 75,A -37.1261,B 24.8998,C -2.3106,E1 25.1361,E2 121.4535} C_DIS
LIN {X 61.794,Y -36.3814,Z 75,A -35.5303,B 24.8998,C -2.3109,E1 25.1384,E2 119.865} C_DIS
LIN {X 63.6918,Y -32.948,Z 75,A -32.1536,B 24.8984,C -2.327,E1 25.1429,E2 116.4682} C_DIS
LIN {X 65.1513,Y -29.9586,Z 75,A -29.5688,B 24.8979,C -2.3327,E1 25.146,E2 113.8837} C_DIS
LIN {X 66.3881,Y -27.1057,Z 75,A -27.3947,B 24.898,C -2.3313,E1 25.1484,E2 111.725} C_DIS
LIN {X 67.6356,Y -23.8229,Z 75,A -24.4069,B 24.8968,C -2.3451,E1 25.1513,E2 108.7212} C_DIS
LIN {X 68.3974,Y -21.5406,Z 75,A -22.3446,B 24.8959,C -2.355,E1 25.153,E2 106.647} C_DIS
LIN {X 69.32,Y -18.3564,Z 75,A -19.874,B 24.8957,C -2.3581,E1 25.1549,E2 104.1833} C_DIS
LIN {X 69.9564,Y -15.759,Z 75,A -17.6967,B 24.895,C -2.366,E1 25.1563,E2 102} C_DIS
LIN {X 70.4861,Y -13.1891,Z 75,A -15.682,B 24.8946,C -2.3703,E1 25.1573,E2 99.9871} C_DIS
LIN {X 70.9544,Y -10.3758,Z 75,A -13.4384,B 24.894,C -2.3765,E1 25.1583,E2 97.742} C_DIS
LIN {X 71.2785,Y -7.8502,Z 75,A -10.8176,B 24.8919,C -2.4,E1 25.1592,E2 95.0812} C_DIS
LIN {X 71.6771,Y -2.1194,Z 75,A -6.7615,B 24.8919,C -2.399,E1 25.1598,E2 91.0515} C_DIS
LIN {X 71.7009,Y 1.0665,Z 75,A -4.4739,B 24.8919,C -2.3996,E1 25.1598,E2 88.776} C_DIS
LIN {X 71.6027,Y 3.8935,Z 75,A -1.9497,B 24.8906,C -2.4144,E1 25.1594,E2 86.2319} C_DIS
LIN {X 71.3399,Y 7.2579,Z 75,A 0.8854,B 24.8895,C -2.4269,E1 25.1587,E2 83.384} C_DIS
LIN {X 70.9297,Y 10.5426,Z 75,A 3.3562,B 24.8892,C -2.4301,E1 25.1578,E2 80.9203} C_DIS
LIN {X 70.39,Y 13.6881,Z 75,A 5.9119,B 24.8884,C -2.4381,E1 25.1565,E2 78.3606} C_DIS
LIN {X 69.6867,Y 16.9075,Z 75,A 8.3307,B 24.8883,C -2.44,E1 25.155,E2 75.9514} C_DIS
LIN {X 69.0547,Y 19.3286,Z 75,A 10.4665,B 24.8874,C -2.4499,E1 25.1534,E2 73.8045} C_DIS
LIN {X 68.1213,Y 22.3986,Z 75,A 13.0967,B 24.8865,C -2.4594,E1 25.1512,E2 71.1668} C_DIS
LIN {X 66.9885,Y 25.5866,Z 75,A 15.2918,B 24.8871,C -2.4527,E1 25.1491,E2 68.9996} C_DIS
LIN {X 65.2389,Y 29.7674,Z 75,A 19.3811,B 24.8849,C -2.4763,E1 25.1446,E2 64.8771} C_DIS
LIN {X 63.7495,Y 32.8351,Z 75,A 21.8234,B 24.8849,C -2.4757,E1 25.1415,E2 62.4491} C_DIS
LIN {X 62.464,Y 35.2198,Z 75,A 24.1112,B 24.8841,C -2.485,E1 25.1384,E2 60.1514} C_DIS
LIN {X 61.1536,Y 37.4486,Z 75,A 26.212,B 24.8835,C -2.4914,E1 25.1354,E2 58.0462} C_DIS
LIN {X 59.5887,Y 39.8927,Z 75,A 28.5406,B 24.8829,C -2.4976,E1 25.1318,E2 55.7147} C_DIS
LIN {X 57.7316,Y 42.5347,Z 75,A 31.0243,B 24.8826,C -2.5012,E1 25.1278,E2 53.2345} C_DIS
LIN {X 55.7724,Y 45.0727,Z 75,A 33.4574,B 24.8823,C -2.5037,E1 25.1236,E2 50.8069} C_DIS
LIN {X 54.1729,Y 46.9836,Z 75,A 36.0829,B 24.8802,C -2.5259,E1 25.1187,E2 48.1407} C_DIS
LIN {X 50.2155,Y 51.191,Z 75,A 39.788,B 24.8817,C -2.5105,E1 25.1117,E2 44.4879} C_DIS
LIN {X 48.3621,Y 52.9455,Z 75,A 42.1919,B 24.8804,C -2.5246,E1 25.1067,E2 42.0605} C_DIS
LIN {X 46.327,Y 54.7353,Z 75,A 44.2652,B 24.8802,C -2.5263,E1 25.1023,E2 39.9915} C_DIS
LIN {X 44.2328,Y 56.4415,Z 75,A 46.7442,B 24.879,C -2.539,E1 25.0969,E2 37.4916} C_DIS
LIN {X 41.5735,Y 58.4273,Z 75,A 49.1774,B 24.8791,C -2.5375,E1 25.0914,E2 35.0704} C_DIS
LIN {X 39.3255,Y 59.9636,Z 75,A 51.3347,B 24.8788,C -2.5405,E1 25.0864,E2 32.9133} C_DIS
LIN {X 36.9174,Y 61.4764,Z 75,A 53.6551,B 24.8784,C -2.5451,E1 25.0808,E2 30.5892} C_DIS
LIN {X 33.9939,Y 63.1392,Z 75,A 56.3035,B 24.8781,C -2.5478,E1 25.0744,E2 27.9423} C_DIS
LIN {X 31.2071,Y 64.5619,Z 75,A 59.4773,B 24.8761,C -2.5689,E1 25.0663,E2 24.7267} C_DIS
LIN {X 28.0905,Y 65.9779,Z 75,A 61.2807,B 24.8782,C -2.547,E1 25.0618,E2 22.9797} C_DIS
LIN {X 25.66,Y 66.9607,Z 75,A 63.5216,B 24.8777,C -2.5529,E1 25.056,E2 20.7297} C_DIS
LIN {X 23.2253,Y 67.8439,Z 75,A 65.7358,B 24.8771,C -2.5585,E1 25.0501,E2 18.5068} C_DIS
LIN {X 20.2817,Y 68.7805,Z 75,A 68.1101,B 24.8771,C -2.5579,E1 25.0438,E2 16.1381} C_DIS
LIN {X 17.4041,Y 69.5656,Z 75,A 70.546,B 24.8769,C -2.5607,E1 25.0372,E2 13.6994} C_DIS
LIN {X 14.5754,Y 70.2117,Z 75,A 72.8442,B 24.8769,C -2.5613,E1 25.031,E2 11.4028} C_DIS
LIN {X 11.2345,Y 70.8235,Z 75,A 75.4028,B 24.8771,C -2.5582,E1 25.0239,E2 8.8541} C_DIS
LIN {X 8.8706,Y 71.1585,Z 75,A 77.2904,B 24.8771,C -2.5582,E1 25.0187,E2 6.9683} C_DIS
LIN {X 6.3321,Y 71.4288,Z 75,A 79.5059,B 24.8767,C -2.5628,E1 25.0125,E2 4.7429} C_DIS
LIN {X 3.1936,Y 71.6373,Z 75,A 81.98,B 24.8767,C -2.5618,E1 25.0056,E2 2.2722} C_DIS
LIN {X 0.0682,Y 71.7093,Z 75,A 84.4546,B 24.8769,C -2.5608,E1 24.9987,E2 -0.1998} C_DIS
LIN {X -2.8668,Y 71.6514,Z 75,A 86.8048,B 24.8769,C -2.5603,E1 24.9922,E2 -2.5489} C_DIS
LIN {X -6.1175,Y 71.4481,Z 75,A 89.4641,B 24.8769,C -2.5605,E1 24.9848,E2 -5.21} C_DIS
LIN {X -8.8941,Y 71.1554,Z 75,A 91.6638,B 24.8771,C -2.5585,E1 24.9787,E2 -7.4064} C_DIS
LIN {X -11.2767,Y 70.8167,Z 75,A 93.7587,B 24.8768,C -2.5615,E1 24.9729,E2 -9.5101} C_DIS
LIN {X -14.7895,Y 70.1677,Z 75,A 96.4498,B 24.8774,C -2.5552,E1 24.9655,E2 -12.1892} C_DIS
LIN {X -17.725,Y 69.4834,Z 75,A 98.7687,B 24.8779,C -2.5507,E1 24.9593,E2 -14.5008} C_DIS
LIN {X -19.5556,Y 68.9904,Z 75,A 101.0464,B 24.8762,C -2.5678,E1 24.953,E2 -16.8227} C_DIS
LIN {X -22.6947,Y 68.0228,Z 75,A 102.9871,B 24.8781,C -2.548,E1 24.948,E2 -18.72} C_DIS
LIN {X -25.188,Y 67.1395,Z 75,A 105.2086,B 24.8781,C -2.548,E1 24.9422,E2 -20.9458} C_DIS
LIN {X -29.864,Y 65.1953,Z 75,A 109.0629,B 24.8791,C -2.5376,E1 24.9323,E2 -24.7843} C_DIS
LIN {X -33.0284,Y 63.6507,Z 75,A 112.0906,B 24.8791,C -2.5382,E1 24.9247,E2 -27.8215} C_DIS
LIN {X -35.8139,Y 62.1246,Z 75,A 114.5204,B 24.8797,C -2.5313,E1 24.9188,E2 -30.2419} C_DIS
LIN {X -38.4338,Y 60.5398,Z 75,A 116.9976,B 24.8801,C -2.5275,E1 24.913,E2 -32.7178} C_DIS
LIN {X -40.7154,Y 59.029,Z 75,A 119.2118,B 24.8804,C -2.5239,E1 24.9078,E2 -34.9309} C_DIS
LIN {X -43.1506,Y 57.2724,Z 75,A 121.5929,B 24.8809,C -2.5186,E1 24.9025,E2 -37.3078} C_DIS
LIN {X -45.3988,Y 55.5081,Z 75,A 123.9079,B 24.8813,C -2.5144,E1 24.8975,E2 -39.6216} C_DIS
LIN {X -47.522,Y 53.7022,Z 75,A 126.159,B 24.8817,C -2.51,E1 24.8927,E2 -41.871} C_DIS
LIN {X -49.5706,Y 51.8163,Z 75,A 128.2821,B 24.8824,C -2.5026,E1 24.8884,E2 -43.9849} C_DIS
LIN {X -51.3418,Y 50.0628,Z 75,A 130.4852,B 24.8824,C -2.5026,E1 24.8841,E2 -46.1976} C_DIS
LIN {X -53.6181,Y 47.616,Z 75,A 133.044,B 24.8833,C -2.4935,E1 24.8793,E2 -48.7459} C_DIS
LIN {X -55.381,Y 45.554,Z 75,A 135.2457,B 24.8837,C -2.4887,E1 24.8753,E2 -50.9463} C_DIS
LIN {X -57.0853,Y 43.399,Z 75,A 137.8581,B 24.8834,C -2.4925,E1 24.8709,E2 -53.5801} C_DIS
LIN {X -59.5158,Y 40.0003,Z 75,A 140.8306,B 24.885,C -2.4751,E1 24.8662,E2 -56.5257} C_DIS
LIN {X -61.1887,Y 37.3907,Z 75,A 143.347,B 24.8856,C -2.4691,E1 24.8624,E2 -59.0406} C_DIS
LIN {X -62.7814,Y 34.6515,Z 75,A 145.8613,B 24.8863,C -2.4614,E1 24.859,E2 -61.5498} C_DIS
LIN {X -64.704,Y 30.9113,Z 75,A 149.2128,B 24.8872,C -2.4514,E1 24.8548,E2 -64.8954} C_DIS
LIN {X -65.9569,Y 28.1404,Z 75,A 151.5151,B 24.8881,C -2.4413,E1 24.8522,E2 -67.1863} C_DIS
LIN {X -67.8174,Y 23.3013,Z 75,A 155.5596,B 24.8895,C -2.4265,E1 24.8483,E2 -71.2182} C_DIS
LIN {X -68.7567,Y 20.362,Z 75,A 158.7977,B 24.8886,C -2.4362,E1 24.8456,E2 -74.4979} C_DIS
LIN {X -69.6773,Y 16.9461,Z 75,A 161.5589,B 24.8896,C -2.4259,E1 24.8437,E2 -77.2507} C_DIS
LIN {X -70.5313,Y 12.9419,Z 75,A 164.5256,B 24.8911,C -2.4088,E1 24.8421,E2 -80.194} C_DIS
LIN {X -71.0085,Y 9.995,Z 75,A 166.9195,B 24.8918,C -2.4014,E1 24.8411,E2 -82.5847} C_DIS
LIN {X -71.3863,Y 6.7921,Z 75,A 169.4994,B 24.8925,C -2.3933,E1 24.8403,E2 -85.1606} C_DIS
LIN {X -71.6248,Y 3.485,Z 75,A 172.1929,B 24.8932,C -2.3859,E1 24.8399,E2 -87.8525} C_DIS
LIN {X -71.7073,Y 0.4905,Z 75,A 174.5634,B 24.8939,C -2.3778,E1 24.8398,E2 -90.218} C_DIS
LIN {X -71.666,Y -2.4814,Z 75,A 176.9806,B 24.8945,C -2.3712,E1 24.8399,E2 -92.634} C_DIS
LIN {X -71.5006,Y -5.4609,Z 75,A 179.0458,B 24.8958,C -2.3566,E1 24.8403,E2 -94.6769} C_DIS
LIN {X -71.2738,Y -7.8946,Z 75,A -178.9071,B 24.8961,C -2.3526,E1 24.8409,E2 -96.7266} C_DIS
LIN {X -70.953,Y -10.3851,Z 75,A -176.5989,B 24.8961,C -2.3531,E1 24.8418,E2 -99.0498} C_DIS
LIN {X -70.4559,Y -13.3459,Z 75,A -174.217,B 24.8968,C -2.3453,E1 24.8429,E2 -101.4272} C_DIS
LIN {X -69.7288,Y -16.7352,Z 75,A -171.0935,B 24.8968,C -2.3449,E1 24.8449,E2 -104.5679} C_DIS
LIN {X -68.5595,Y -21.0178,Z 75,A -167.8877,B 24.8984,C -2.3266,E1 24.8474,E2 -107.7486} C_DIS
LIN {X -67.6888,Y -23.6712,Z 75,A -165.111,B 24.8979,C -2.3324,E1 24.8499,E2 -110.5551} C_DIS
LIN {X -66.134,Y -27.7203,Z 75,A -162.1871,B 24.8999,C -2.3102,E1 24.8529,E2 -113.4421} C_DIS
LIN {X -64.8506,Y -30.6045,Z 75,A -159.5777,B 24.9003,C -2.3051,E1 24.8559,E2 -116.0537} C_DIS
LIN {X -62.9457,Y -34.3506,Z 75,A -156.2146,B 24.9011,C -2.2961,E1 24.8603,E2 -119.4133} C_DIS
LIN {X -61.4457,Y -36.9678,Z 75,A -153.7817,B 24.9016,C -2.2903,E1 24.8637,E2 -121.845} C_DIS
LIN {X -60.2875,Y -38.8269,Z 75,A -151.7967,B 24.9016,C -2.2913,E1 24.8667,E2 -123.8423} C_DIS
LIN {X -58.3766,Y -41.6446,Z 75,A -149.2789,B 24.9025,C -2.2798,E1 24.8707,E2 -126.3453} C_DIS
LIN {X -56.7633,Y -43.8181,Z 75,A -147.2312,B 24.9032,C -2.272,E1 24.8742,E2 -128.384} C_DIS
LIN {X -55.114,Y -45.8753,Z 75,A -144.9699,B 24.9032,C -2.2707,E1 24.8782,E2 -130.6528} C_DIS
LIN {X -53.0801,Y -48.2155,Z 75,A -142.4632,B 24.9037,C -2.2659,E1 24.8828,E2 -133.1592} C_DIS
LIN {X -50.8615,Y -50.5495,Z 75,A -139.9046,B 24.9042,C -2.2601,E1 24.8878,E2 -135.715} C_DIS
LIN {X -48.5749,Y -52.7502,Z 75,A -137.4565,B 24.9048,C -2.253,E1 24.8928,E2 -138.1561} C_DIS
LIN {X -46.3311,Y -54.7318,Z 75,A -135.2996,B 24.9056,C -2.2428,E1 24.8973,E2 -140.2973} C_DIS
LIN {X -44.5073,Y -56.2245,Z 75,A -133.202,B 24.9055,C -2.2445,E1 24.9019,E2 -142.4067} C_DIS
LIN {X -42.1169,Y -58.0375,Z 75,A -130.7058,B 24.9056,C -2.2428,E1 24.9075,E2 -144.9077} C_DIS
LIN {X -40.0098,Y -59.5094,Z 75,A -128.7508,B 24.9061,C -2.2371,E1 24.912,E2 -146.8558} C_DIS
LIN {X -37.6104,Y -61.055,Z 75,A -126.2544,B 24.906,C -2.2389,E1 24.9179,E2 -149.3643} C_DIS
LIN {X -34.8007,Y -62.698,Z 75,A -123.9169,B 24.9068,C -2.2289,E1 24.9235,E2 -151.685} C_DIS
LIN {X -31.0215,Y -64.6511,Z 75,A -120.2189,B 24.9065,C -2.232,E1 24.9328,E2 -155.4003} C_DIS
LIN {X -28.2316,Y -65.9181,Z 75,A -117.8511,B 24.9069,C -2.2274,E1 24.9388,E2 -157.7628} C_DIS
LIN {X -25.7009,Y -66.9452,Z 75,A -115.7299,B 24.9072,C -2.2239,E1 24.9443,E2 -159.8801} C_DIS
LIN {X -23.4251,Y -67.7752,Z 75,A -113.7279,B 24.9072,C -2.2239,E1 24.9496,E2 -161.8861} C_DIS
LIN {X -20.8302,Y -68.6169,Z 75,A -111.5435,B 24.9073,C -2.2224,E1 24.9554,E2 -164.0708} C_DIS
LIN {X -17.7939,Y -69.4656,Z 75,A -109.1295,B 24.9077,C -2.2183,E1 24.9619,E2 -166.4786} C_DIS
LIN {X -16.0598,Y -69.8869,Z 75,A -106.5525,B 24.9053,C -2.2469,E1 24.9692,E2 -169.127} C_DIS
LIN {X -11.858,Y -70.7212,Z 75,A -104.1565,B 24.9076,C -2.2194,E1 24.9756,E2 -171.4601} C_DIS
LIN {X -7.3243,Y -71.3335,Z 75,A -99.9701,B 24.9065,C -2.2326,E1 24.9873,E2 -175.6804} C_DIS
LIN {X -2.7691,Y -71.6556,Z 75,A -97.0852,B 24.9081,C -2.2129,E1 24.9952,E2 -178.5196} C_DIS
LIN {X -0.042,Y -71.7095,Z 75,A -94.6362,B 24.9075,C -2.2203,E1 25.0021,E2 -180.9862} C_DIS
LIN {X -0.042,Y -71.7095,Z 75,A -94.6362,B 24.9075,C -2.2203,E1 25.0021,E2 -180.9862} C_DIS
Enddeposition()
LIN {X 0.4691,Y -70.8074,Z 75,A -95.8047,B 24.9096,C -2.1959,E1 24.9987,E2 -179.7597} C_DIS
Startdeposition()
$VEL.CP = VEL_PRINT
LIN {X -3.3665,Y -70.7297,Z 75,A -98.6771,B 24.9091,C -2.2013,E1 24.9907,E2 -176.8997} C_DIS
LIN {X -7.3091,Y -70.4308,Z 75,A -102.0022,B 24.9093,C -2.1983,E1 24.9814,E2 -173.5659} C_DIS
LIN {X -10.6952,Y -69.9967,Z 75,A -104.707,B 24.9092,C -2.2004,E1 24.9739,E2 -170.8637} C_DIS
LIN {X -15.9684,Y -68.985,Z 75,A -108.2698,B 24.9074,C -2.2213,E1 24.9643,E2 -167.3467} C_DIS
LIN {X -18.0344,Y -68.4751,Z 75,A -110.6849,B 24.9088,C -2.2053,E1 24.9576,E2 -164.8901} C_DIS
LIN {X -21.089,Y -67.5957,Z 75,A -113.2128,B 24.9085,C -2.2082,E1 24.9509,E2 -162.3647} C_DIS
LIN {X -24.7898,Y -66.3285,Z 75,A -116.0012,B 24.9076,C -2.2199,E1 24.9436,E2 -159.5987} C_DIS
LIN {X -27.969,Y -65.0521,Z 75,A -119.7598,B 24.9093,C -2.1992,E1 24.9338,E2 -155.7824} C_DIS
LIN {X -33.1975,Y -62.5451,Z 75,A -123.6486,B 24.9072,C -2.2238,E1 24.9242,E2 -151.9419} C_DIS
LIN {X -35.5002,Y -61.2675,Z 75,A -126.027,B 24.9075,C -2.2209,E1 24.9183,E2 -149.5496} C_DIS
LIN {X -39.1719,Y -58.9875,Z 75,A -129.4929,B 24.907,C -2.2269,E1 24.9102,E2 -146.087} C_DIS
LIN {X -41.7015,Y -57.227,Z 75,A -131.9439,B 24.9065,C -2.232,E1 24.9046,E2 -143.6396} C_DIS
LIN {X -44.8368,Y -54.8058,Z 75,A -135.0731,B 24.9059,C -2.2395,E1 24.8978,E2 -140.5167} C_DIS
LIN {X -46.4854,Y -53.4138,Z 75,A -137.0864,B 24.9062,C -2.2367,E1 24.8935,E2 -138.4889} C_DIS
LIN {X -48.7706,Y -51.3368,Z 75,A -139.482,B 24.9055,C -2.244,E1 24.8886,E2 -136.101} C_DIS
LIN {X -51.2992,Y -48.8106,Z 75,A -142.1029,B 24.9045,C -2.2562,E1 24.8835,E2 -133.498} C_DIS
LIN {X -52.9615,Y -47.0009,Z 75,A -144.2918,B 24.9045,C -2.2561,E1 24.8794,E2 -131.2991} C_DIS
LIN {X -54.7986,Y -44.8457,Z 75,A -146.9324,B 24.9047,C -2.2535,E1 24.8746,E2 -128.6402} C_DIS
LIN {X -56.8419,Y -42.2262,Z 75,A -149.5056,B 24.904,C -2.2625,E1 24.8703,E2 -126.0761} C_DIS
LIN {X -58.6094,Y -39.7347,Z 75,A -152.5918,B 24.9046,C -2.2552,E1 24.8654,E2 -122.9571} C_DIS
LIN {X -60.4621,Y -36.8546,Z 75,A -155.227,B 24.9037,C -2.2653,E1 24.8616,E2 -120.3326} C_DIS
LIN {X -63.1752,Y -31.9824,Z 75,A -159.3016,B 24.9019,C -2.287,E1 24.8562,E2 -116.2881} C_DIS
LIN {X -64.417,Y -29.4019,Z 75,A -161.518,B 24.9011,C -2.2956,E1 24.8536,E2 -114.0802} C_DIS
LIN {X -65.6355,Y -26.5691,Z 75,A -164.7005,B 24.9018,C -2.2879,E1 24.8502,E2 -110.8616} C_DIS
LIN {X -66.7852,Y -23.5295,Z 75,A -166.4651,B 24.8995,C -2.3142,E1 24.8486,E2 -109.1499} C_DIS
LIN {X -67.9761,Y -19.8283,Z 75,A -169.8327,B 24.8991,C -2.3187,E1 24.8458,E2 -105.7736} C_DIS
LIN {X -68.5264,Y -17.8351,Z 75,A -172.4051,B 24.9004,C -2.3045,E1 24.844,E2 -103.1523} C_DIS
LIN {X -69.3804,Y -14.1522,Z 75,A -174.3245,B 24.8974,C -2.3382,E1 24.8429,E2 -101.3021} C_DIS
LIN {X -69.7942,Y -11.9479,Z 75,A -177.336,B 24.8992,C -2.3182,E1 24.8414,E2 -98.225} C_DIS
LIN {X -70.3379,Y -8.1545,Z 75,A -179.2645,B 24.8961,C -2.3529,E1 24.8408,E2 -96.3678} C_DIS
LIN {X -70.6114,Y -5.297,Z 75,A 178.3793,B 24.8955,C -2.3594,E1 24.8402,E2 -94.0131} C_DIS
LIN {X -70.7432,Y -3.0518,Z 75,A 176.3731,B 24.8954,C -2.3612,E1 24.8399,E2 -91.9989} C_DIS
LIN {X -70.8108,Y 0.0899,Z 75,A 173.6364,B 24.895,C -2.365,E1 24.8398,E2 -89.2549} C_DIS
LIN {X -70.7279,Y 3.4072,Z 75,A 170.7485,B 24.8947,C -2.3692,E1 24.8401,E2 -86.3598} C_DIS
LIN {X -70.4519,Y 7.1074,Z 75,A 167.9493,B 24.8934,C -2.3831,E1 24.8408,E2 -83.5769} C_DIS
LIN {X -70.0571,Y 10.2969,Z 75,A 165.3308,B 24.8927,C -2.391,E1 24.8418,E2 -80.9615} C_DIS
LIN {X -69.5237,Y 13.43,Z 75,A 162.8172,B 24.8919,C -2.4003,E1 24.843,E2 -78.4553} C_DIS
LIN {X -68.7777,Y 16.8388,Z 75,A 159.9988,B 24.8911,C -2.4093,E1 24.8447,E2 -75.6418} C_DIS
LIN {X -67.8997,Y 20.0883,Z 75,A 157.0202,B 24.8908,C -2.4123,E1 24.847,E2 -72.6531} C_DIS
LIN {X -66.8009,Y 23.4853,Z 75,A 153.5268,B 24.8912,C -2.4083,E1 24.8502,E2 -69.1303} C_DIS
LIN {X -65.5771,Y 26.7126,Z 75,A 151.614,B 24.8887,C -2.4355,E1 24.8521,E2 -67.2717} C_DIS
LIN {X -64.2069,Y 29.8562,Z 75,A 148.863,B 24.8879,C -2.4442,E1 24.8552,E2 -64.5265} C_DIS
LIN {X -62.4283,Y 33.4181,Z 75,A 144.8417,B 24.8886,C -2.4364,E1 24.8605,E2 -60.465} C_DIS
LIN {X -60.141,Y 37.3764,Z 75,A 140.8528,B 24.8882,C -2.4406,E1 24.8663,E2 -56.4657} C_DIS
LIN {X -58.0998,Y 40.4762,Z 75,A 138.8926,B 24.8854,C -2.4713,E1 24.8693,E2 -54.5691} C_DIS
LIN {X -56.9273,Y 42.1099,Z 75,A 136.5643,B 24.8864,C -2.4604,E1 24.8732,E2 -52.2035} C_DIS
LIN {X -54.0301,Y 45.7678,Z 75,A 133.2413,B 24.8846,C -2.48,E1 24.879,E2 -48.9119} C_DIS
LIN {X -51.8652,Y 48.2088,Z 75,A 130.1664,B 24.8848,C -2.477,E1 24.8848,E2 -45.8162} C_DIS
LIN {X -48.4241,Y 51.6627,Z 75,A 127.0445,B 24.8823,C -2.5045,E1 24.8909,E2 -42.7468} C_DIS
LIN {X -46.9464,Y 53.0103,Z 75,A 124.9698,B 24.8829,C -2.498,E1 24.8953,E2 -40.6482} C_DIS
LIN {X -44.6275,Y 54.9755,Z 75,A 122.6297,B 24.8821,C -2.506,E1 24.9003,E2 -38.3184} C_DIS
LIN {X -41.8899,Y 57.089,Z 75,A 119.1406,B 24.883,C -2.4964,E1 24.9082,E2 -34.7938} C_DIS
LIN {X -38.3804,Y 59.5053,Z 75,A 116.2429,B 24.8812,C -2.5153,E1 24.9148,E2 -31.9317} C_DIS
LIN {X -35.6596,Y 61.1757,Z 75,A 113.5668,B 24.881,C -2.5178,E1 24.9212,E2 -29.2534} C_DIS
LIN {X -31.0306,Y 63.6488,Z 75,A 109.1875,B 24.8806,C -2.5217,E1 24.9321,E2 -24.8714} C_DIS
LIN {X -26.753,Y 65.5606,Z 75,A 105.2593,B 24.8804,C -2.524,E1 24.9422,E2 -20.9396} C_DIS
LIN {X -22.86,Y 67.017,Z 75,A 102.0242,B 24.8797,C -2.5312,E1 24.9507,E2 -17.7151} C_DIS
LIN {X -18.8881,Y 68.2447,Z 75,A 98.883,B 24.8789,C -2.54,E1 24.959,E2 -14.5897} C_DIS
LIN {X -16.1816,Y 68.9357,Z 75,A 96.4344,B 24.8791,C -2.5377,E1 24.9657,E2 -12.1322} C_DIS
LIN {X -11.9049,Y 69.8012,Z 75,A 92.8175,B 24.8791,C -2.5384,E1 24.9756,E2 -8.5132} C_DIS
LIN {X -8.2995,Y 70.3209,Z 75,A 90.2243,B 24.8781,C -2.5487,E1 24.9827,E2 -5.9425} C_DIS
LIN {X -5.4135,Y 70.6021,Z 75,A 87.7516,B 24.8782,C -2.5467,E1 24.9896,E2 -3.4639} C_DIS
LIN {X -1.0203,Y 70.8022,Z 75,A 84.4109,B 24.8776,C -2.5531,E1 24.9989,E2 -0.1378} C_DIS
LIN {X 1.2915,Y 70.7972,Z 75,A 82.309,B 24.8781,C -2.5478,E1 25.0048,E2 1.9766} C_DIS
LIN {X 4.3681,Y 70.6753,Z 75,A 79.8124,B 24.8781,C -2.5478,E1 25.0118,E2 4.4724} C_DIS
LIN {X 7.5639,Y 70.4041,Z 75,A 76.9557,B 24.8788,C -2.541,E1 25.0198,E2 7.3433} C_DIS
LIN {X 11.4183,Y 69.8828,Z 75,A 74.0963,B 24.8782,C -2.5473,E1 25.0276,E2 10.1853} C_DIS
LIN {X 14.5008,Y 69.3088,Z 75,A 71.4702,B 24.8785,C -2.544,E1 25.0348,E2 12.816} C_DIS
LIN {X 17.6497,Y 68.5741,Z 75,A 68.7837,B 24.8788,C -2.5408,E1 25.0421,E2 15.5062} C_DIS
LIN {X 21.7093,Y 67.399,Z 75,A 65.7966,B 24.878,C -2.5493,E1 25.05,E2 18.468} C_DIS
LIN {X 23.8483,Y 66.6734,Z 75,A 63.6199,B 24.879,C -2.5388,E1 25.0558,E2 20.6652} C_DIS
LIN {X 27.9013,Y 65.0816,Z 75,A 59.608,B 24.8805,C -2.5227,E1 25.0663,E2 24.7058} C_DIS
LIN {X 31.0011,Y 63.663,Z 75,A 57.3843,B 24.8795,C -2.5332,E1 25.0718,E2 26.899} C_DIS
LIN {X 33.8734,Y 62.1813,Z 75,A 54.623,B 24.8802,C -2.526,E1 25.0786,E2 29.6696} C_DIS
LIN {X 37.0924,Y 60.3175,Z 75,A 51.805,B 24.8802,C -2.5266,E1 25.0854,E2 32.4774} C_DIS
LIN {X 39.4477,Y 58.8038,Z 75,A 49.5708,B 24.8804,C -2.5239,E1 25.0906,E2 34.7108} C_DIS
LIN {X 43.5988,Y 55.7961,Z 75,A 45.6985,B 24.8804,C -2.5239,E1 25.0993,E2 38.5689} C_DIS
LIN {X 46.2159,Y 53.6484,Z 75,A 42.7344,B 24.8815,C -2.5129,E1 25.1056,E2 41.548} C_DIS
LIN {X 48.548,Y 51.5462,Z 75,A 40.3291,B 24.8816,C -2.5115,E1 25.1106,E2 43.9469} C_DIS
LIN {X 50.2454,Y 49.8933,Z 75,A 38.0293,B 24.8829,C -2.4972,E1 25.1152,E2 46.2708} C_DIS
LIN {X 53.31,Y 46.6043,Z 75,A 34.5764,B 24.8832,C -2.4941,E1 25.1216,E2 49.7156} C_DIS
LIN {X 55.1912,Y 44.3613,Z 75,A 31.6587,B 24.8851,C -2.4738,E1 25.1268,E2 52.6678} C_DIS
LIN {X 57.7559,Y 40.9659,Z 75,A 28.8001,B 24.8844,C -2.4812,E1 25.1315,E2 55.4951} C_DIS
LIN {X 59.4502,Y 38.4662,Z 75,A 26.4667,B 24.8847,C -2.478,E1 25.1351,E2 57.8245} C_DIS
LIN {X 61.036,Y 35.8963,Z 75,A 23.6198,B 24.8864,C -2.4606,E1 25.1392,E2 60.6979} C_DIS
LIN {X 62.8247,Y 32.6667,Z 75,A 20.9013,B 24.8864,C -2.4599,E1 25.1428,E2 63.4038} C_DIS
LIN {X 64.3347,Y 29.5816,Z 75,A 18.1145,B 24.8872,C -2.452,E1 25.1461,E2 66.1944} C_DIS
LIN {X 66.1158,Y 25.3515,Z 75,A 14.6919,B 24.8874,C -2.4494,E1 25.1497,E2 69.6041} C_DIS
LIN {X 67.0134,Y 22.8733,Z 75,A 12.4825,B 24.8882,C -2.4411,E1 25.1517,E2 71.8208} C_DIS
LIN {X 68.1304,Y 19.2913,Z 75,A 9.4009,B 24.8891,C -2.4308,E1 25.1542,E2 74.9091} C_DIS
LIN {X 68.7006,Y 17.1547,Z 75,A 7.6158,B 24.8896,C -2.4255,E1 25.1555,E2 76.6965} C_DIS
LIN {X 69.3579,Y 14.2616,Z 75,A 5.2354,B 24.8902,C -2.4187,E1 25.1569,E2 79.079} C_DIS
LIN {X 69.9011,Y 11.3085,Z 75,A 2.7805,B 24.891,C -2.4105,E1 25.158,E2 81.539} C_DIS
LIN {X 70.2925,Y 8.5399,Z 75,A 0.1106,B 24.8926,C -2.3921,E1 25.159,E2 84.2366} C_DIS
LIN {X 70.6716,Y 4.4223,Z 75,A -2.6975,B 24.8922,C -2.3965,E1 25.1596,E2 87.0174} C_DIS
LIN {X 70.8033,Y 0.9609,Z 75,A -5.8412,B 24.8939,C -2.3781,E1 25.1598,E2 90.186} C_DIS
LIN {X 70.7579,Y -2.7085,Z 75,A -8.8497,B 24.8948,C -2.3676,E1 25.1595,E2 93.2014} C_DIS
LIN {X 70.3901,Y -7.6972,Z 75,A -12.0908,B 24.8939,C -2.3774,E1 25.1588,E2 96.4002} C_DIS
LIN {X 69.9377,Y -11.0772,Z 75,A -15.3868,B 24.8961,C -2.3535,E1 25.1575,E2 99.7331} C_DIS
LIN {X 69.3404,Y -14.3467,Z 75,A -17.8833,B 24.8963,C -2.3505,E1 25.1561,E2 102.2222} C_DIS
LIN {X 68.6566,Y -17.3285,Z 75,A -20.3863,B 24.8971,C -2.3419,E1 25.1545,E2 104.731} C_DIS
LIN {X 67.3802,Y -21.7674,Z 75,A -23.9511,B 24.8977,C -2.3352,E1 25.1517,E2 108.2914} C_DIS
LIN {X 65.9466,Y -25.787,Z 75,A -27.8191,B 24.8996,C -2.3131,E1 25.1479,E2 112.19} C_DIS
LIN {X 63.8996,Y -30.5088,Z 75,A -31.7678,B 24.9002,C -2.3066,E1 25.1433,E2 116.1324} C_DIS
LIN {X 62.5357,Y -33.2153,Z 75,A -33.9187,B 24.9001,C -2.3079,E1 25.1406,E2 118.2691} C_DIS
LIN {X 60.8557,Y -36.2014,Z 75,A -36.6275,B 24.9006,C -2.3017,E1 25.1368,E2 120.9784} C_DIS
LIN {X 59.5593,Y -38.2963,Z 75,A -38.8076,B 24.9015,C -2.2909,E1 25.1336,E2 123.173} C_DIS
LIN {X 57.9163,Y -40.7403,Z 75,A -41.4618,B 24.9027,C -2.2769,E1 25.1293,E2 125.8473} C_DIS
LIN {X 55.7264,Y -43.6871,Z 75,A -43.741,B 24.9018,C -2.2881,E1 25.1255,E2 128.0891} C_DIS
LIN {X 54.3701,Y -45.3632,Z 75,A -45.8747,B 24.9031,C -2.2728,E1 25.1217,E2 130.2491} C_DIS
LIN {X 52.3401,Y -47.6916,Z 75,A -48.2987,B 24.9034,C -2.2686,E1 25.1172,E2 132.6723} C_DIS
LIN {X 50.0241,Y -50.1162,Z 75,A -51.1213,B 24.9043,C -2.259,E1 25.1117,E2 135.5054} C_DIS
LIN {X 47.5966,Y -52.427,Z 75,A -53.7397,B 24.9046,C -2.2553,E1 25.1063,E2 138.122} C_DIS
LIN {X 45.2583,Y -54.4573,Z 75,A -56.0928,B 24.9047,C -2.2538,E1 25.1013,E2 140.4694} C_DIS
LIN {X 43.5805,Y -55.8106,Z 75,A -57.7005,B 24.9047,C -2.2538,E1 25.0978,E2 142.0712} C_DIS
LIN {X 41.5791,Y -57.3165,Z 75,A -60.0615,B 24.9058,C -2.2405,E1 25.0925,E2 144.4551} C_DIS
LIN {X 39.6319,Y -58.679,Z 75,A -61.7971,B 24.9058,C -2.2418,E1 25.0885,E2 146.1818} C_DIS
LIN {X 37.1637,Y -60.2739,Z 75,A -64.3136,B 24.9064,C -2.2335,E1 25.0825,E2 148.7097} C_DIS
LIN {X 34.5058,Y -61.8325,Z 75,A -66.7784,B 24.9067,C -2.2299,E1 25.0766,E2 151.1757} C_DIS
LIN {X 31.5878,Y -63.3731,Z 75,A -70.3062,B 24.909,C -2.2029,E1 25.0676,E2 154.7579} C_DIS
LIN {X 28.0293,Y -65.0258,Z 75,A -72.4601,B 24.9071,C -2.225,E1 25.0623,E2 156.8543} C_DIS
LIN {X 23.3815,Y -66.8373,Z 75,A -76.8926,B 24.9084,C -2.2092,E1 25.0506,E2 161.3147} C_DIS
LIN {X 20.158,Y -67.8791,Z 75,A -79.9041,B 24.9093,C -2.1991,E1 25.0425,E2 164.3448} C_DIS
LIN {X 15.6619,Y -69.0558,Z 75,A -83.103,B 24.9084,C -2.2099,E1 25.0339,E2 167.5135} C_DIS
LIN {X 12.5731,Y -69.6838,Z 75,A -85.617,B 24.9084,C -2.2087,E1 25.027,E2 170.0273} C_DIS
LIN {X 8.8172,Y -70.2584,Z 75,A -88.751,B 24.9088,C -2.2051,E1 25.0183,E2 173.167} C_DIS
LIN {X 5.6768,Y -70.5811,Z 75,A -91.1163,B 24.9085,C -2.2086,E1 25.0118,E2 175.5226} C_DIS
LIN {X 3.0298,Y -70.7441,Z 75,A -93.2773,B 24.9085,C -2.2074,E1 25.0058,E2 177.6858} C_DIS
LIN {X 0.4691,Y -70.8074,Z 75,A -94.4579,B 24.9068,C -2.2295,E1 25.0026,E2 178.8138} C_DIS
Enddeposition()
LIN {X 0.4691,Y -70.8074,Z 75,A -94.4579,B 24.9068,C -2.2295,E1 25.0026,E2 178.8138} C_DIS
Startdeposition()
$VEL.CP = VEL_PRINT
LIN {X 1.3932,Y -69.8958,Z 75,A -93.6041,B 24.9052,C -2.2476,E1 25.0051,E2 177.9171} C_DIS
LIN {X 4.3264,Y -69.7766,Z 75,A -91.1698,B 24.9051,C -2.2493,E1 25.0119,E2 175.4797} C_DIS
LIN {X 7.193,Y -69.5386,Z 75,A -88.6096,B 24.9045,C -2.2557,E1 25.0191,E2 172.9057} C_DIS
LIN {X 11.5288,Y -68.9524,Z 75,A -85.1951,B 24.9047,C -2.2538,E1 25.0285,E2 169.4989} C_DIS
LIN {X 14.5745,Y -68.3743,Z 75,A -82.6537,B 24.9045,C -2.2559,E1 25.0354,E2 166.9556} C_DIS
LIN {X 16.4931,Y -67.9362,Z 75,A -79.9095,B 24.9018,C -2.2874,E1 25.0431,E2 164.1408} C_DIS
LIN {X 20.8807,Y -66.7187,Z 75,A -77.3577,B 24.9042,C -2.2603,E1 25.0497,E2 161.6577} C_DIS
LIN {X 24.7929,Y -65.3656,Z 75,A -73.6036,B 24.903,C -2.2743,E1 25.0596,E2 157.8783} C_DIS
LIN {X 27.7326,Y -64.174,Z 75,A -71.4528,B 24.9037,C -2.2661,E1 25.0651,E2 155.752} C_DIS
LIN {X 31.4579,Y -62.4332,Z 75,A -67.6684,B 24.9023,C -2.2825,E1 25.0747,E2 151.9388} C_DIS
LIN {X 35.0238,Y -60.5039,Z 75,A -64.7434,B 24.9027,C -2.2776,E1 25.0818,E2 149.034} C_DIS
LIN {X 37.5819,Y -58.9491,Z 75,A -62.318,B 24.9024,C -2.2814,E1 25.0875,E2 146.6073} C_DIS
LIN {X 41.0011,Y -56.625,Z 75,A -58.5352,B 24.9008,C -2.2989,E1 25.0962,E2 142.796} C_DIS
LIN {X 43.9608,Y -54.3581,Z 75,A -55.8424,B 24.9011,C -2.2956,E1 25.1021,E2 140.1211} C_DIS
LIN {X 46.3912,Y -52.3001,Z 75,A -53.2213,B 24.9006,C -2.3017,E1 25.1076,E2 137.4958} C_DIS
LIN {X 49.3649,Y -49.5031,Z 75,A -49.6695,B 24.8994,C -2.3153,E1 25.1148,E2 133.9267} C_DIS
LIN {X 51.9105,Y -46.8264,Z 75,A -46.8968,B 24.8994,C -2.3158,E1 25.12,E2 131.165} C_DIS
LIN {X 54.01,Y -44.3893,Z 75,A -44.4335,B 24.8992,C -2.3178,E1 25.1244,E2 128.7083} C_DIS
LIN {X 55.9812,Y -41.8744,Z 75,A -41.2203,B 24.8971,C -2.3413,E1 25.13,E2 125.4547} C_DIS
LIN {X 58.3455,Y -38.5117,Z 75,A -38.327,B 24.8975,C -2.3372,E1 25.1345,E2 122.5853} C_DIS
LIN {X 59.9161,Y -36.021,Z 75,A -35.2284,B 24.8952,C -2.3633,E1 25.139,E2 119.4408} C_DIS
LIN {X 61.5758,Y -33.103,Z 75,A -33.3449,B 24.8967,C -2.3468,E1 25.1415,E2 117.6062} C_DIS
LIN {X 63.2305,Y -29.8199,Z 75,A -30.2281,B 24.8956,C -2.3586,E1 25.1453,E2 114.4782} C_DIS
LIN {X 64.2275,Y -27.6097,Z 75,A -27.6651,B 24.8936,C -2.3808,E1 25.1482,E2 111.8768} C_DIS
LIN {X 66.2387,Y -22.3558,Z 75,A -24.2284,B 24.8953,C -2.3618,E1 25.1515,E2 108.5042} C_DIS
LIN {X 67.6096,Y -17.7891,Z 75,A -19.7616,B 24.8928,C -2.3896,E1 25.155,E2 103.9973} C_DIS
LIN {X 68.2796,Y -15.0084,Z 75,A -17.7199,B 24.893,C -2.3884,E1 25.1563,E2 101.9701} C_DIS
LIN {X 69.0129,Y -11.1659,Z 75,A -14.0615,B 24.8909,C -2.4113,E1 25.1581,E2 98.2792} C_DIS
LIN {X 69.4709,Y -7.8256,Z 75,A -11.2141,B 24.8899,C -2.4225,E1 25.1591,E2 95.4223} C_DIS
LIN {X 69.8322,Y -3.3018,Z 75,A -8.0233,B 24.8902,C -2.4193,E1 25.1597,E2 92.2578} C_DIS
LIN {X 69.8998,Y 1.1748,Z 75,A -3.6351,B 24.8872,C -2.4513,E1 25.1597,E2 87.8202} C_DIS
LIN {X 69.6603,Y 5.9079,Z 75,A -0.2138,B 24.8873,C -2.4504,E1 25.159,E2 84.4213} C_DIS
LIN {X 69.2728,Y 9.4234,Z 75,A 3.0137,B 24.8856,C -2.4687,E1 25.1579,E2 81.1696} C_DIS
LIN {X 68.5446,Y 13.7509,Z 75,A 6.1297,B 24.8858,C -2.4662,E1 25.1563,E2 78.0777} C_DIS
LIN {X 67.8334,Y 16.9144,Z 75,A 9.1226,B 24.8842,C -2.4837,E1 25.1543,E2 75.0607} C_DIS
LIN {X 66.0908,Y 22.7923,Z 75,A 13.7958,B 24.8837,C -2.4887,E1 25.1505,E2 70.4022} C_DIS
LIN {X 64.8813,Y 26.0331,Z 75,A 16.6679,B 24.8829,C -2.4979,E1 25.1476,E2 67.5243} C_DIS
LIN {X 63.4292,Y 29.3956,Z 75,A 19.6458,B 24.8821,C -2.5057,E1 25.1442,E2 64.5443} C_DIS
LIN {X 62.1592,Y 31.9942,Z 75,A 22.0132,B 24.8815,C -2.5121,E1 25.1412,E2 62.1743} C_DIS
LIN {X 60.4597,Y 35.1009,Z 75,A 25.0028,B 24.8806,C -2.5222,E1 25.1371,E2 59.1763} C_DIS
LIN {X 58.5698,Y 38.1715,Z 75,A 27.773,B 24.8803,C -2.5247,E1 25.1329,E2 56.4142} C_DIS
LIN {X 57.3008,Y 40.0499,Z 75,A 29.9107,B 24.8792,C -2.537,E1 25.1295,E2 54.2578} C_DIS
LIN {X 54.3744,Y 43.9407,Z 75,A 33.3596,B 24.8797,C -2.5317,E1 25.1236,E2 50.8378} C_DIS
LIN {X 52.3057,Y 46.385,Z 75,A 36.8231,B 24.8769,C -2.5605,E1 25.1172,E2 47.3218} C_DIS
LIN {X 50.1062,Y 48.7526,Z 75,A 38.9408,B 24.8778,C -2.5517,E1 25.1131,E2 45.234} C_DIS
LIN {X 47.3779,Y 51.4072,Z 75,A 41.9875,B 24.8773,C -2.5561,E1 25.107,E2 42.1895} C_DIS
LIN {X 44.9529,Y 53.5416,Z 75,A 44.8169,B 24.8764,C -2.566,E1 25.1009,E2 39.3476} C_DIS
LIN {X 42.9644,Y 55.1502,Z 75,A 47.0219,B 24.8757,C -2.5727,E1 25.0961,E2 37.1351} C_DIS
LIN {X 38.4094,Y 58.4129,Z 75,A 51.2202,B 24.876,C -2.5697,E1 25.0865,E2 32.9581} C_DIS
LIN {X 36.0254,Y 59.9135,Z 75,A 54.1434,B 24.8741,C -2.5894,E1 25.0794,E2 29.9975} C_DIS
LIN {X 31.7984,Y 62.2592,Z 75,A 57.4564,B 24.8753,C -2.5775,E1 25.0713,E2 26.722} C_DIS
LIN {X 29.9262,Y 63.1816,Z 75,A 59.1348,B 24.8752,C -2.5787,E1 25.0671,E2 25.0452} C_DIS
LIN {X 27.7116,Y 64.1831,Z 75,A 61.4148,B 24.8742,C -2.5883,E1 25.0612,E2 22.7478} C_DIS
LIN {X 23.3968,Y 65.8787,Z 75,A 64.9068,B 24.8746,C -2.584,E1 25.0522,E2 19.2737} C_DIS
LIN {X 18.681,Y 67.368,Z 75,A 69.0783,B 24.8741,C -2.5899,E1 25.041,E2 15.0954} C_DIS
LIN {X 15.4388,Y 68.1842,Z 75,A 71.7609,B 24.8741,C -2.5899,E1 25.0337,E2 12.4166} C_DIS
LIN {X 12.5465,Y 68.7747,Z 75,A 74.1244,B 24.8741,C -2.5895,E1 25.0273,E2 10.0568} C_DIS
LIN {X 10.6466,Y 69.0941,Z 75,A 76.4138,B 24.8723,C -2.6078,E1 25.0208,E2 7.7261} C_DIS
LIN {X 7.3682,Y 69.5202,Z 75,A 78.7632,B 24.8732,C -2.5992,E1 25.0144,E2 5.3988} C_DIS
LIN {X 3.433,Y 69.8264,Z 75,A 81.7024,B 24.8739,C -2.5919,E1 25.0062,E2 2.4783} C_DIS
LIN {X 0.2046,Y 69.9096,Z 75,A 84.0771,B 24.8746,C -2.5848,E1 24.9996,E2 0.1206} C_DIS
LIN {X -5.119,Y 69.7231,Z 75,A 88.701,B 24.8741,C -2.5896,E1 24.9867,E2 -4.5156} C_DIS
LIN {X -8.1158,Y 69.4369,Z 75,A 91.145,B 24.8743,C -2.5877,E1 24.9799,E2 -6.9566} C_DIS
LIN {X -12.539,Y 68.7761,Z 75,A 94.858,B 24.8744,C -2.5863,E1 24.9697,E2 -10.6696} C_DIS
LIN {X -15.9543,Y 68.0651,Z 75,A 97.8921,B 24.8743,C -2.588,E1 24.9614,E2 -13.7116} C_DIS
LIN {X -18.5354,Y 67.4083,Z 75,A 100.3368,B 24.8739,C -2.592,E1 24.9548,E2 -16.1695} C_DIS
LIN {X -23.575,Y 65.8156,Z 75,A 104.1446,B 24.8756,C -2.5745,E1 24.9448,E2 -19.9427} C_DIS
LIN {X -26.5592,Y 64.6684,Z 75,A 107.14,B 24.8751,C -2.5797,E1 24.937,E2 -22.9571} C_DIS
LIN {X -31.2477,Y 62.5378,Z 75,A 111.0695,B 24.8763,C -2.5665,E1 24.9271,E2 -26.8651} C_DIS
LIN {X -33.512,Y 61.3542,Z 75,A 113.5075,B 24.8759,C -2.5709,E1 24.9211,E2 -29.3205} C_DIS
LIN {X -38.0647,Y 58.6392,Z 75,A 117.8939,B 24.8766,C -2.5639,E1 24.9107,E2 -33.7039} C_DIS
LIN {X -41.8286,Y 56.0157,Z 75,A 121.2814,B 24.8781,C -2.5479,E1 24.903,E2 -37.065} C_DIS
LIN {X -44.5215,Y 53.9001,Z 75,A 124.1767,B 24.8785,C -2.5439,E1 24.8967,E2 -39.9616} C_DIS
LIN {X -46.8172,Y 51.9188,Z 75,A 126.3367,B 24.8797,C -2.531,E1 24.8922,E2 -42.0995} C_DIS
LIN {X -49.7474,Y 49.1176,Z 75,A 130.0958,B 24.8796,C -2.5329,E1 24.8847,E2 -45.8788} C_DIS
LIN {X -52.4626,Y 46.2072,Z 75,A 133.2512,B 24.8806,C -2.5225,E1 24.8788,E2 -49.0233} C_DIS
LIN {X -54.2196,Y 44.1317,Z 75,A 136.55,B 24.8788,C -2.5406,E1 24.8729,E2 -52.3806} C_DIS
LIN {X -56.7672,Y 40.8031,Z 75,A 138.5679,B 24.8827,C -2.5,E1 24.8697,E2 -54.3115} C_DIS
LIN {X -58.181,Y 38.7609,Z 75,A 141.3709,B 24.8816,C -2.5113,E1 24.8652,E2 -57.1552} C_DIS
LIN {X -59.9049,Y 36.0396,Z 75,A 143.7197,B 24.8829,C -2.4975,E1 24.8618,E2 -59.4831} C_DIS
LIN {X -61.6985,Y 32.8734,Z 75,A 147.0812,B 24.8829,C -2.4972,E1 24.8573,E2 -62.8617} C_DIS
LIN {X -63.1106,Y 30.0741,Z 75,A 149.9614,B 24.883,C -2.4964,E1 24.8538,E2 -65.7557} C_DIS
LIN {X -64.4579,Y 27.0654,Z 75,A 151.7549,B 24.8856,C -2.4686,E1 24.8519,E2 -67.4926} C_DIS
LIN {X -65.781,Y 23.67,Z 75,A 155.3707,B 24.8852,C -2.4731,E1 24.8483,E2 -71.1396} C_DIS
LIN {X -67.1497,Y 19.4487,Z 75,A 159.2325,B 24.8858,C -2.4668,E1 24.8452,E2 -75.0085} C_DIS
LIN {X -68.798,Y 12.4168,Z 75,A 164.0594,B 24.8897,C -2.4246,E1 24.8423,E2 -79.763} C_DIS
LIN {X -69.1775,Y 10.0942,Z 75,A 166.5207,B 24.8892,C -2.4299,E1 24.8412,E2 -82.2516} C_DIS
LIN {X -69.5425,Y 7.1559,Z 75,A 168.663,B 24.8904,C -2.4161,E1 24.8405,E2 -84.3738} C_DIS
LIN {X -69.831,Y 3.3294,Z 75,A 172.5132,B 24.89,C -2.4213,E1 24.8399,E2 -88.2596} C_DIS
LIN {X -69.9098,Y -0.3127,Z 75,A 175.1579,B 24.8915,C -2.4045,E1 24.8399,E2 -90.8799} C_DIS
LIN {X -69.8313,Y -3.322,Z 75,A 177.4773,B 24.8925,C -2.3935,E1 24.84,E2 -93.1871} C_DIS
LIN {X -69.5124,Y -7.4433,Z 75,A -179.3494,B 24.8939,C -2.3783,E1 24.8408,E2 -96.3431} C_DIS
LIN {X -69.0968,Y -10.629,Z 75,A -175.7421,B 24.8927,C -2.3912,E1 24.8422,E2 -100.0028} C_DIS
LIN {X -68.0659,Y -15.948,Z 75,A -171.5782,B 24.8945,C -2.3716,E1 24.8446,E2 -104.1443} C_DIS
LIN {X -67.1118,Y -19.5759,Z 75,A -168.3781,B 24.895,C -2.3652,E1 24.847,E2 -107.3476} C_DIS
LIN {X -66.164,Y -22.5774,Z 75,A -165.8694,B 24.8958,C -2.356,E1 24.8492,E2 -109.8487} C_DIS
LIN {X -64.5268,Y -26.9018,Z 75,A -162.2773,B 24.8972,C -2.3408,E1 24.8529,E2 -113.4246} C_DIS
LIN {X -63.3608,Y -29.5424,Z 75,A -159.4235,B 24.8968,C -2.345,E1 24.8563,E2 -116.3041} C_DIS
LIN {X -61.4982,Y -33.2465,Z 75,A -156.5791,B 24.8987,C -2.3235,E1 24.8599,E2 -119.1123} C_DIS
LIN {X -59.6883,Y -36.3959,Z 75,A -153.7443,B 24.8997,C -2.3125,E1 24.8639,E2 -121.9356} C_DIS
LIN {X -57.908,Y -39.1664,Z 75,A -150.7803,B 24.8997,C -2.3116,E1 24.8684,E2 -124.9123} C_DIS
LIN {X -56.1027,Y -41.7127,Z 75,A -148.3839,B 24.9006,C -2.3017,E1 24.8723,E2 -127.2968} C_DIS
LIN {X -53.5541,Y -44.938,Z 75,A -144.9746,B 24.9012,C -2.2948,E1 24.8783,E2 -130.7054} C_DIS
LIN {X -50.9866,Y -47.8301,Z 75,A -142.1588,B 24.9025,C -2.2798,E1 24.8835,E2 -133.498} C_DIS
LIN {X -48.6529,Y -50.2024,Z 75,A -138.9736,B 24.9021,C -2.2844,E1 24.8898,E2 -136.7079} C_DIS
LIN {X -45.7731,Y -52.8418,Z 75,A -135.9362,B 24.903,C -2.2744,E1 24.8961,E2 -139.7335} C_DIS
LIN {X -43.7764,Y -54.5075,Z 75,A -133.4147,B 24.9025,C -2.2795,E1 24.9016,E2 -142.2767} C_DIS
LIN {X -39.3324,Y -57.7956,Z 75,A -128.1449,B 24.9017,C -2.2894,E1 24.9137,E2 -147.5882} C_DIS
LIN {X -36.2246,Y -59.7924,Z 75,A -125.9043,B 24.9036,C -2.2663,E1 24.9189,E2 -149.7808} C_DIS
LIN {X -33.3851,Y -61.423,Z 75,A -123.4911,B 24.9045,C -2.2563,E1 24.9247,E2 -152.1772} C_DIS
LIN {X -30.639,Y -62.8392,Z 75,A -120.4258,B 24.9037,C -2.2659,E1 24.9325,E2 -155.2734} C_DIS
LIN {X -25.8872,Y -64.9409,Z 75,A -116.6979,B 24.9051,C -2.2487,E1 24.942,E2 -158.9691} C_DIS
LIN {X -21.8101,Y -66.4211,Z 75,A -112.6349,B 24.9043,C -2.258,E1 24.9527,E2 -163.0622} C_DIS
LIN {X -18.179,Y -67.5046,Z 75,A -109.8599,B 24.9052,C -2.2479,E1 24.9601,E2 -165.8177} C_DIS
LIN {X -15.8769,Y -68.083,Z 75,A -107.4621,B 24.9043,C -2.2581,E1 24.9667,E2 -168.2429} C_DIS
LIN {X -12.019,Y -68.8696,Z 75,A -104.57,B 24.9051,C -2.2486,E1 24.9746,E2 -171.1155} C_DIS
LIN {X -8.6799,Y -69.3689,Z 75,A -101.357,B 24.9042,C -2.2592,E1 24.9836,E2 -174.3562} C_DIS
LIN {X -3.3927,Y -69.8283,Z 75,A -97.5584,B 24.9054,C -2.2453,E1 24.9941,E2 -178.1233} C_DIS
LIN {X 0.4744,Y -69.8905,Z 75,A -95.5803,B 24.9079,C -2.2164,E1 24.9994,E2 -180.0327} C_DIS
Enddeposition()
LIN {X 0.4744,Y -69.8905,Z 75,A -95.5803,B 24.9079,C -2.2164,E1 24.9994,E2 -180.0327} C_DIS
Startdeposition()
$VEL.CP = VEL_PRINT
Enddeposition()
END
